LIN {X 0,Y 698.249,Z 977.53,A -85,B 0,C 180,E1 3562.598,E2 3562.598} C_VEL
LIN {X 0,Y 698.325,Z 977.53,A -85,B 0,C 180,E1 3567.816,E2 3567.816} C_VEL
LIN {X 0,Y 698.444,Z 977.53,A -85,B 0,C 180,E1 3572.91,E2 3572.91} C_VEL
LIN {X 0,Y 698.552,Z 977.53,A -85,B 0,C 180,E1 3577.03,E2 3577.03} C_VEL
LIN {X 0,Y 698.572,Z 977.53,A -85,B 0,C 180,E1 3582.649,E2 3582.649} C_VEL
LIN {X 0,Y 698.411,Z 977.53,A -85,B 0,C 180,E1 3587.531,E2 3587.531} C_VEL
LIN {X 0,Y 698.656,Z 977.53,A -85,B 0,C 180,E1 3592.533,E2 3592.533} C_VEL
LIN {X 0,Y 698.798,Z 977.53,A -85,B 0,C 180,E1 3596.63,E2 3596.63} C_VEL
LIN {X 0,Y 700.664,Z 990.787,A -85,B 0,C 180,E1 3596.832,E2 3596.832} C_VEL
LIN {X 0,Y 700.6,Z 1043.986,A -85,B 0,C 180,E1 3597.491,E2 3597.491} C_VEL
LIN {X 0,Y 700.227,Z 1071.881,A -85,B 0,C 180,E1 3598.304,E2 3598.304} C_VEL
LIN {X 0,Y 699.823,Z 1097.341,A -85,B 0,C 180,E1 3599.544,E2 3599.544} C_VEL
LIN {X 0,Y 699.493,Z 1119.031,A -85,B 0,C 180,E1 3601.095,E2 3601.095} C_VEL
LIN {X 0,Y 699.241,Z 1137.078,A -85,B 0,C 180,E1 3602.959,E2 3602.959} C_VEL
LIN {X 0,Y 699.113,Z 1150.198,A -85,B 0,C 180,E1 3604.982,E2 3604.982} C_VEL
LIN {X 0,Y 699.023,Z 1157.754,A -85,B 0,C 180,E1 3606.855,E2 3606.855} C_VEL
LIN {X 0,Y 698.935,Z 1161.69,A -85,B 0,C 180,E1 3608.737,E2 3608.737} C_VEL
LIN {X 0,Y 698.932,Z 1161.598,A -85,B 0,C 180,E1 3611.259,E2 3611.259} C_VEL
LIN {X 0,Y 699.047,Z 1156.293,A -85,B 0,C 180,E1 3613.499,E2 3613.499} C_VEL
LIN {X 0,Y 699.09,Z 1145.799,A -85,B 0,C 180,E1 3615.702,E2 3615.702} C_VEL
LIN {X 0,Y 699.304,Z 1129.473,A -85,B 0,C 180,E1 3617.829,E2 3617.829} C_VEL
LIN {X 0,Y 699.637,Z 1108.274,A -85,B 0,C 180,E1 3619.654,E2 3619.654} C_VEL
LIN {X 0,Y 700.068,Z 1082.113,A -85,B 0,C 180,E1 3621.168,E2 3621.168} C_VEL
LIN {X 0,Y 700.436,Z 1054.54,A -85,B 0,C 180,E1 3622.169,E2 3622.169} C_VEL
LIN {X 0,Y 700.63,Z 1024.887,A -85,B 0,C 180,E1 3622.707,E2 3622.707} C_VEL
LIN {X 0,Y 699.655,Z 981.842,A -85,B 0,C 180,E1 3623.185,E2 3623.185} C_VEL
LIN {X 0,Y 698.753,Z 977.53,A -85,B 0,C 180,E1 3623.298,E2 3623.298} C_VEL
LIN {X 0,Y 698.38,Z 977.53,A -85,B 0,C 180,E1 3628.518,E2 3628.518} C_VEL
LIN {X 0,Y 698.358,Z 977.53,A -85,B 0,C 180,E1 3632.856,E2 3632.856} C_VEL
LIN {X 0,Y 698.369,Z 977.53,A -85,B 0,C 180,E1 3637.416,E2 3637.416} C_VEL
LIN {X 0,Y 698.407,Z 977.53,A -85,B 0,C 180,E1 3642.459,E2 3642.459} C_VEL
LIN {X 0,Y 698.22,Z 977.53,A -85,B 0,C 180,E1 3647.712,E2 3647.712} C_VEL
LIN {X 0,Y 698.256,Z 977.53,A -85,B 0,C 180,E1 3652.575,E2 3652.575} C_VEL
LIN {X 0,Y 698.326,Z 977.53,A -85,B 0,C 180,E1 3657.811,E2 3657.811} C_VEL
LIN {X 0,Y 698.438,Z 977.53,A -85,B 0,C 180,E1 3662.89,E2 3662.89} C_VEL
LIN {X 0,Y 698.526,Z 977.53,A -85,B 0,C 180,E1 3667.011,E2 3667.011} C_VEL
LIN {X 0,Y 698.583,Z 977.53,A -85,B 0,C 180,E1 3672.635,E2 3672.635} C_VEL
LIN {X 0,Y 698.447,Z 977.53,A -85,B 0,C 180,E1 3677.502,E2 3677.502} C_VEL
LIN {X 0,Y 698.678,Z 977.53,A -85,B 0,C 180,E1 3682.517,E2 3682.517} C_VEL
LIN {X 0,Y 698.759,Z 977.53,A -85,B 0,C 180,E1 3687.509,E2 3687.509} C_VEL
LIN {X 0,Y 698.622,Z 977.53,A -85,B 0,C 180,E1 3692.48,E2 3692.48} C_VEL
LIN {X 0,Y 698.586,Z 977.53,A -85,B 0,C 180,E1 3696.22,E2 3696.22} C_VEL
LIN {X 0,Y 698.52,Z 977.53,A -85,B 0,C 180,E1 3701.252,E2 3701.252} C_VEL
LIN {X 0,Y 698.586,Z 977.53,A -85,B 0,C 180,E1 3706.372,E2 3706.372} C_VEL
LIN {X 0,Y 698.467,Z 977.53,A -85,B 0,C 180,E1 3711.635,E2 3711.635} C_VEL
LIN {X 0,Y 698.436,Z 977.53,A -85,B 0,C 180,E1 3715.709,E2 3715.709} C_VEL
LIN {X 0,Y 698.354,Z 977.53,A -85,B 0,C 180,E1 3719.93,E2 3719.93} C_VEL
LIN {X 0,Y 698.333,Z 977.53,A -85,B 0,C 180,E1 3724.453,E2 3724.453} C_VEL
LIN {X 0,Y 698.296,Z 977.53,A -85,B 0,C 180,E1 3728.99,E2 3728.99} C_VEL
LIN {X 0,Y 698.43,Z 977.53,A -85,B 0,C 180,E1 3734.274,E2 3734.274} C_VEL
LIN {X 0,Y 698.275,Z 977.53,A -85,B 0,C 180,E1 3739.411,E2 3739.411} C_VEL
LIN {X 0,Y 698.261,Z 977.53,A -85,B 0,C 180,E1 3744.126,E2 3744.126} C_VEL
LIN {X 0,Y 698.368,Z 977.53,A -85,B 0,C 180,E1 3748.612,E2 3748.612} C_VEL
LIN {X 0,Y 698.567,Z 977.53,A -85,B 0,C 180,E1 3754.283,E2 3754.283} C_VEL
LIN {X 0,Y 698.639,Z 977.53,A -85,B 0,C 180,E1 3754.865,E2 3754.865} C_VEL
LIN {X 0,Y 704.591,Z 996.788,A -85,B 0,C 180,E1 3755.324,E2 3755.324} C_VEL
LIN {X 0,Y 704.196,Z 1037.732,A -85,B 0,C 180,E1 3756.085,E2 3756.085} C_VEL
LIN {X 0,Y 703.296,Z 1074.948,A -85,B 0,C 180,E1 3757.243,E2 3757.243} C_VEL
LIN {X 0,Y 702.251,Z 1111.428,A -85,B 0,C 180,E1 3758.889,E2 3758.889} C_VEL
LIN {X 0,Y 701.238,Z 1144.866,A -85,B 0,C 180,E1 3760.94,E2 3760.94} C_VEL
LIN {X 0,Y 700.351,Z 1174.512,A -85,B 0,C 180,E1 3763.334,E2 3763.334} C_VEL
LIN {X 0,Y 699.676,Z 1200.165,A -85,B 0,C 180,E1 3766.051,E2 3766.051} C_VEL
LIN {X 0,Y 699.244,Z 1221.384,A -85,B 0,C 180,E1 3769.062,E2 3769.062} C_VEL
LIN {X 0,Y 699.071,Z 1237.084,A -85,B 0,C 180,E1 3772.206,E2 3772.206} C_VEL
LIN {X 0,Y 698.964,Z 1246.264,A -85,B 0,C 180,E1 3775.017,E2 3775.017} C_VEL
LIN {X 0,Y 698.927,Z 1250.943,A -85,B 0,C 180,E1 3777.506,E2 3777.506} C_VEL
LIN {X 0,Y 698.887,Z 1252.497,A -85,B 0,C 180,E1 3779.991,E2 3779.991} C_VEL
LIN {X 0,Y 698.948,Z 1250.844,A -85,B 0,C 180,E1 3782.476,E2 3782.476} C_VEL
LIN {X 0,Y 699.001,Z 1244.41,A -85,B 0,C 180,E1 3785.588,E2 3785.588} C_VEL
LIN {X 0,Y 699.048,Z 1232.688,A -85,B 0,C 180,E1 3788.717,E2 3788.717} C_VEL
LIN {X 0,Y 699.377,Z 1214.934,A -85,B 0,C 180,E1 3791.867,E2 3791.867} C_VEL
LIN {X 0,Y 699.823,Z 1192.335,A -85,B 0,C 180,E1 3794.772,E2 3794.772} C_VEL
LIN {X 0,Y 696.246,Z 1182.329,A -85,B 0,C 180,E1 3795.917,E2 3795.917} C_VEL
LIN {X 0,Y 692.744,Z 1171.657,A -85,B 0,C 180,E1 3797.032,E2 3797.032} C_VEL
LIN {X 0,Y 693.801,Z 1140.2,A -85,B 0,C 180,E1 3799.52,E2 3799.52} C_VEL
LIN {X 0,Y 694.966,Z 1105.397,A -85,B 0,C 180,E1 3801.576,E2 3801.576} C_VEL
LIN {X 0,Y 696.116,Z 1067.835,A -85,B 0,C 180,E1 3803.183,E2 3803.183} C_VEL
LIN {X 0,Y 697.047,Z 1028.121,A -85,B 0,C 180,E1 3804.317,E2 3804.317} C_VEL
LIN {X 0,Y 696.867,Z 995.477,A -85,B 0,C 180,E1 3804.895,E2 3804.895} C_VEL
LIN {X 0,Y 690.399,Z 977.53,A -85,B 0,C 180,E1 3805.41,E2 3805.41} C_VEL
LIN {X 0,Y 690.4,Z 977.53,A -85,B 0,C 180,E1 3810.303,E2 3810.303} C_VEL
LIN {X 0,Y 690.417,Z 977.53,A -85,B 0,C 180,E1 3815.714,E2 3815.714} C_VEL
LIN {X 0,Y 690.242,Z 977.53,A -85,B 0,C 180,E1 3819.804,E2 3819.804} C_VEL
LIN {X 0,Y 690.201,Z 977.53,A -85,B 0,C 180,E1 3824.611,E2 3824.611} C_VEL
LIN {X 0,Y 690.209,Z 977.53,A -85,B 0,C 180,E1 3828.814,E2 3828.814} C_VEL
LIN {X 0,Y 690.525,Z 977.53,A -85,B 0,C 180,E1 3834.259,E2 3834.259} C_VEL
LIN {X 0,Y 690.336,Z 977.53,A -85,B 0,C 180,E1 3839.686,E2 3839.686} C_VEL
LIN {X 0,Y 690.417,Z 977.584,A -85,B 0,C 180,E1 3842.029,E2 3842.029} C_VEL
LIN {X 0,Y 694.054,Z 987.272,A -85,B 0,C 180,E1 3842.718,E2 3842.718} C_VEL
LIN {X 0,Y 700.633,Z 994.826,A -85,B 0,C 180,E1 3843.899,E2 3843.899} C_VEL
LIN {X 0,Y 700.298,Z 999.146,A -85,B 0,C 180,E1 3844.205,E2 3844.205} C_VEL
LIN {X 0,Y 697.744,Z 1009.008,A -85,B 0,C 180,E1 3844.567,E2 3844.567} C_VEL
LIN {X 0,Y 697.181,Z 1078.924,A -85,B 0,C 180,E1 3845.446,E2 3845.446} C_VEL
LIN {X 0,Y 696.429,Z 1117.843,A -85,B 0,C 180,E1 3846.435,E2 3846.435} C_VEL
LIN {X 0,Y 695.282,Z 1155.762,A -85,B 0,C 180,E1 3847.911,E2 3847.911} C_VEL
LIN {X 0,Y 694.12,Z 1191.102,A -85,B 0,C 180,E1 3849.839,E2 3849.839} C_VEL
LIN {X 0,Y 692.969,Z 1223.117,A -85,B 0,C 180,E1 3852.18,E2 3852.18} C_VEL
LIN {X 0,Y 692.08,Z 1250.219,A -85,B 0,C 180,E1 3854.774,E2 3854.774} C_VEL
LIN {X 0,Y 691.534,Z 1273.012,A -85,B 0,C 180,E1 3857.67,E2 3857.67} C_VEL
LIN {X 0,Y 691.198,Z 1289.555,A -85,B 0,C 180,E1 3860.48,E2 3860.48} C_VEL
LIN {X 0,Y 691.049,Z 1302.604,A -85,B 0,C 180,E1 3863.712,E2 3863.712} C_VEL
LIN {X 0,Y 691.004,Z 1308.965,A -85,B 0,C 180,E1 3866.234,E2 3866.234} C_VEL
LIN {X 0,Y 691.014,Z 1312.108,A -85,B 0,C 180,E1 3868.749,E2 3868.749} C_VEL
LIN {X 0,Y 690.994,Z 1312.099,A -85,B 0,C 180,E1 3871.262,E2 3871.262} C_VEL
LIN {X 0,Y 691.006,Z 1307.534,A -85,B 0,C 180,E1 3874.464,E2 3874.464} C_VEL
LIN {X 0,Y 691.174,Z 1296.933,A -85,B 0,C 180,E1 3877.881,E2 3877.881} C_VEL
LIN {X 0,Y 691.431,Z 1281.1,A -85,B 0,C 180,E1 3881.061,E2 3881.061} C_VEL
LIN {X 0,Y 691.888,Z 1259.84,A -85,B 0,C 180,E1 3884.108,E2 3884.108} C_VEL
LIN {X 0,Y 692.673,Z 1234.009,A -85,B 0,C 180,E1 3886.855,E2 3886.855} C_VEL
LIN {X 0,Y 693.688,Z 1204.373,A -85,B 0,C 180,E1 3889.271,E2 3889.271} C_VEL
LIN {X 0,Y 694.806,Z 1170.678,A -85,B 0,C 180,E1 3891.348,E2 3891.348} C_VEL
LIN {X 0,Y 695.991,Z 1133.36,A -85,B 0,C 180,E1 3893.029,E2 3893.029} C_VEL
LIN {X 0,Y 696.975,Z 1094.227,A -85,B 0,C 180,E1 3894.224,E2 3894.224} C_VEL
LIN {X 0,Y 697.524,Z 1054.281,A -85,B 0,C 180,E1 3894.928,E2 3894.928} C_VEL
LIN {X 0,Y 697.79,Z 1008.208,A -85,B 0,C 180,E1 3895.492,E2 3895.492} C_VEL
LIN {X 0,Y 700.714,Z 996.51,A -85,B 0,C 180,E1 3895.944,E2 3895.944} C_VEL
LIN {X 0,Y 698.106,Z 991.717,A -85,B 0,C 180,E1 3896.672,E2 3896.672} C_VEL
LIN {X 0,Y 692.741,Z 985.09,A -85,B 0,C 180,E1 3897.48,E2 3897.48} C_VEL
LIN {X 0,Y 690.418,Z 977.53,A -85,B 0,C 180,E1 3898.047,E2 3898.047} C_VEL
LIN {X 0,Y 690.399,Z 977.53,A -85,B 0,C 180,E1 3903.284,E2 3903.284} C_VEL
LIN {X 0,Y 690.433,Z 977.53,A -85,B 0,C 180,E1 3907.923,E2 3907.923} C_VEL
LIN {X 0,Y 690.497,Z 977.53,A -85,B 0,C 180,E1 3913.62,E2 3913.62} C_VEL
LIN {X 0,Y 690.271,Z 977.53,A -85,B 0,C 180,E1 3918.828,E2 3918.828} C_VEL
LIN {X 0,Y 690.331,Z 977.53,A -85,B 0,C 180,E1 3924.316,E2 3924.316} C_VEL
LIN {X 0,Y 690.414,Z 977.53,A -85,B 0,C 180,E1 3929.697,E2 3929.697} C_VEL
LIN {X 0,Y 690.611,Z 977.53,A -85,B 0,C 180,E1 3934.116,E2 3934.116} C_VEL
LIN {X 0,Y 690.58,Z 977.53,A -85,B 0,C 180,E1 3939.459,E2 3939.459} C_VEL
LIN {X 0,Y 690.604,Z 977.53,A -85,B 0,C 180,E1 3944.746,E2 3944.746} C_VEL
LIN {X 0,Y 690.737,Z 977.53,A -85,B 0,C 180,E1 3949.903,E2 3949.903} C_VEL
LIN {X 0,Y 690.735,Z 977.53,A -85,B 0,C 180,E1 3954.976,E2 3954.976} C_VEL
LIN {X 0,Y 690.849,Z 977.53,A -85,B 0,C 180,E1 3956.418,E2 3956.418} C_VEL
LIN {X 0,Y 693.134,Z 991.243,A -85,B 0,C 180,E1 3956.645,E2 3956.645} C_VEL
LIN {X 0,Y 693.015,Z 1044.752,A -85,B 0,C 180,E1 3957.324,E2 3957.324} C_VEL
LIN {X 0,Y 692.601,Z 1073.222,A -85,B 0,C 180,E1 3958.168,E2 3958.168} C_VEL
LIN {X 0,Y 692.165,Z 1099.161,A -85,B 0,C 180,E1 3959.46,E2 3959.46} C_VEL
LIN {X 0,Y 691.726,Z 1121.136,A -85,B 0,C 180,E1 3961.107,E2 3961.107} C_VEL
LIN {X 0,Y 691.364,Z 1139.428,A -85,B 0,C 180,E1 3963.15,E2 3963.15} C_VEL
LIN {X 0,Y 691.177,Z 1152.174,A -85,B 0,C 180,E1 3965.355,E2 3965.355} C_VEL
LIN {X 0,Y 691.072,Z 1159.704,A -85,B 0,C 180,E1 3967.568,E2 3967.568} C_VEL
LIN {X 0,Y 691.034,Z 1162.385,A -85,B 0,C 180,E1 3970.111,E2 3970.111} C_VEL
LIN {X 0,Y 691.151,Z 1158.995,A -85,B 0,C 180,E1 3972.672,E2 3972.672} C_VEL
LIN {X 0,Y 691.243,Z 1150.473,A -85,B 0,C 180,E1 3974.933,E2 3974.933} C_VEL
LIN {X 0,Y 691.363,Z 1136.614,A -85,B 0,C 180,E1 3977.12,E2 3977.12} C_VEL
LIN {X 0,Y 691.742,Z 1118.326,A -85,B 0,C 180,E1 3979.023,E2 3979.023} C_VEL
LIN {X 0,Y 692.116,Z 1095.401,A -85,B 0,C 180,E1 3980.651,E2 3980.651} C_VEL
LIN {X 0,Y 692.679,Z 1069.013,A -85,B 0,C 180,E1 3981.881,E2 3981.881} C_VEL
LIN {X 0,Y 692.893,Z 1040.067,A -85,B 0,C 180,E1 3982.663,E2 3982.663} C_VEL
LIN {X 0,Y 692.216,Z 983.619,A -85,B 0,C 180,E1 3983.346,E2 3983.346} C_VEL
LIN {X 0,Y 690.826,Z 977.53,A -85,B 0,C 180,E1 3983.517,E2 3983.517} C_VEL
LIN {X 0,Y 690.461,Z 977.53,A -85,B 0,C 180,E1 3988.875,E2 3988.875} C_VEL
LIN {X 0,Y 690.394,Z 977.53,A -85,B 0,C 180,E1 3993.476,E2 3993.476} C_VEL
LIN {X 0,Y 690.447,Z 977.53,A -85,B 0,C 180,E1 3997.921,E2 3997.921} C_VEL
LIN {X 0,Y 690.507,Z 977.53,A -85,B 0,C 180,E1 4003.593,E2 4003.593} C_VEL
LIN {X 0,Y 690.272,Z 977.53,A -85,B 0,C 180,E1 4008.803,E2 4008.803} C_VEL
LIN {X 0,Y 690.323,Z 977.53,A -85,B 0,C 180,E1 4013.647,E2 4013.647} C_VEL
LIN {X 0,Y 690.434,Z 977.53,A -85,B 0,C 180,E1 4018.867,E2 4018.867} C_VEL
LIN {X 0,Y 690.586,Z 977.53,A -85,B 0,C 180,E1 4024.113,E2 4024.113} C_VEL
LIN {X 0,Y 690.567,Z 977.53,A -85,B 0,C 180,E1 4029.441,E2 4029.441} C_VEL
LIN {X 0,Y 690.654,Z 977.53,A -85,B 0,C 180,E1 4034.88,E2 4034.88} C_VEL
LIN {X 0,Y 690.758,Z 977.53,A -85,B 0,C 180,E1 4039.887,E2 4039.887} C_VEL
LIN {X 0,Y 690.725,Z 977.53,A -85,B 0,C 180,E1 4044.96,E2 4044.96} C_VEL
LIN {X 0,Y 690.796,Z 977.53,A -85,B 0,C 180,E1 4049.994,E2 4049.994} C_VEL
LIN {X 0,Y 690.911,Z 977.53,A -85,B 0,C 180,E1 4055.027,E2 4055.027} C_VEL
LIN {X 0,Y 690.64,Z 977.53,A -85,B 0,C 180,E1 4060.103,E2 4060.103} C_VEL
LIN {X 0,Y 690.634,Z 977.53,A -85,B 0,C 180,E1 4065.259,E2 4065.259} C_VEL
LIN {X 0,Y 690.61,Z 977.53,A -85,B 0,C 180,E1 4070.546,E2 4070.546} C_VEL
LIN {X 0,Y 690.511,Z 977.53,A -85,B 0,C 180,E1 4076.026,E2 4076.026} C_VEL
LIN {X 0,Y 690.44,Z 977.53,A -85,B 0,C 180,E1 4081.134,E2 4081.134} C_VEL
LIN {X 0,Y 690.451,Z 977.53,A -85,B 0,C 180,E1 4086.33,E2 4086.33} C_VEL
LIN {X 0,Y 690.418,Z 977.53,A -85,B 0,C 180,E1 4091.732,E2 4091.732} C_VEL
LIN {X 0,Y 690.369,Z 977.53,A -85,B 0,C 180,E1 4096.402,E2 4096.402} C_VEL
LIN {X 0,Y 690.345,Z 977.53,A -85,B 0,C 180,E1 4102.192,E2 4102.192} C_VEL
LIN {X 0,Y 690.347,Z 977.53,A -85,B 0,C 180,E1 4106.714,E2 4106.714} C_VEL
LIN {X 0,Y 690.468,Z 977.53,A -85,B 0,C 180,E1 4111.368,E2 4111.368} C_VEL
LIN {X 0,Y 690.701,Z 977.53,A -85,B 0,C 180,E1 4114.564,E2 4114.564} C_VEL
LIN {X 0,Y 697.426,Z 998.279,A -85,B 0,C 180,E1 4115.074,E2 4115.074} C_VEL
LIN {X 0,Y 696.954,Z 1038.128,A -85,B 0,C 180,E1 4115.832,E2 4115.832} C_VEL
LIN {X 0,Y 695.918,Z 1075.817,A -85,B 0,C 180,E1 4117.023,E2 4117.023} C_VEL
LIN {X 0,Y 694.785,Z 1111.418,A -85,B 0,C 180,E1 4118.651,E2 4118.651} C_VEL
LIN {X 0,Y 693.641,Z 1145.022,A -85,B 0,C 180,E1 4120.734,E2 4120.734} C_VEL
LIN {X 0,Y 692.632,Z 1174.504,A -85,B 0,C 180,E1 4123.143,E2 4123.143} C_VEL
LIN {X 0,Y 691.853,Z 1200.159,A -85,B 0,C 180,E1 4125.89,E2 4125.89} C_VEL
LIN {X 0,Y 691.393,Z 1221.379,A -85,B 0,C 180,E1 4128.936,E2 4128.936} C_VEL
LIN {X 0,Y 691.176,Z 1237.082,A -85,B 0,C 180,E1 4132.117,E2 4132.117} C_VEL
LIN {X 0,Y 691.059,Z 1246.263,A -85,B 0,C 180,E1 4134.96,E2 4134.96} C_VEL
LIN {X 0,Y 691.048,Z 1250.943,A -85,B 0,C 180,E1 4137.478,E2 4137.478} C_VEL
LIN {X 0,Y 690.989,Z 1252.497,A -85,B 0,C 180,E1 4139.991,E2 4139.991} C_VEL
LIN {X 0,Y 691.07,Z 1250.844,A -85,B 0,C 180,E1 4142.504,E2 4142.504} C_VEL
LIN {X 0,Y 691.11,Z 1244.411,A -85,B 0,C 180,E1 4145.652,E2 4145.652} C_VEL
LIN {X 0,Y 691.175,Z 1232.69,A -85,B 0,C 180,E1 4148.817,E2 4148.817} C_VEL
LIN {X 0,Y 691.536,Z 1214.935,A -85,B 0,C 180,E1 4152.004,E2 4152.004} C_VEL
LIN {X 0,Y 692.059,Z 1192.736,A -85,B 0,C 180,E1 4154.897,E2 4154.897} C_VEL
LIN {X 0,Y 692.744,Z 1171.657,A -85,B 0,C 180,E1 4157.032,E2 4157.032} C_VEL
LIN {X 0,Y 689.415,Z 1160.444,A -85,B 0,C 180,E1 4158.114,E2 4158.114} C_VEL
LIN {X 0,Y 685.964,Z 1148.483,A -85,B 0,C 180,E1 4159.145,E2 4159.145} C_VEL
LIN {X 0,Y 687.188,Z 1114.694,A -85,B 0,C 180,E1 4161.323,E2 4161.323} C_VEL
LIN {X 0,Y 688.488,Z 1078.679,A -85,B 0,C 180,E1 4163.032,E2 4163.032} C_VEL
LIN {X 0,Y 689.598,Z 1040.14,A -85,B 0,C 180,E1 4164.298,E2 4164.298} C_VEL
LIN {X 0,Y 690.337,Z 1001.799,A -85,B 0,C 180,E1 4165.059,E2 4165.059} C_VEL
LIN {X 0,Y 686.176,Z 988.352,A -85,B 0,C 180,E1 4165.395,E2 4165.395} C_VEL
LIN {X 0,Y 682.476,Z 977.53,A -85,B 0,C 180,E1 4165.706,E2 4165.706} C_VEL
LIN {X 0,Y 682.498,Z 977.53,A -85,B 0,C 180,E1 4170.692,E2 4170.692} C_VEL
LIN {X 0,Y 682.505,Z 977.53,A -85,B 0,C 180,E1 4175.241,E2 4175.241} C_VEL
LIN {X 0,Y 682.319,Z 977.53,A -85,B 0,C 180,E1 4180.075,E2 4180.075} C_VEL
LIN {X 0,Y 682.306,Z 977.53,A -85,B 0,C 180,E1 4185.268,E2 4185.268} C_VEL
LIN {X 0,Y 682.316,Z 977.53,A -85,B 0,C 180,E1 4189.915,E2 4189.915} C_VEL
LIN {X 0,Y 682.588,Z 977.53,A -85,B 0,C 180,E1 4195.195,E2 4195.195} C_VEL
LIN {X 0,Y 682.43,Z 977.53,A -85,B 0,C 180,E1 4200.766,E2 4200.766} C_VEL
LIN {X 0,Y 682.52,Z 977.629,A -85,B 0,C 180,E1 4201.762,E2 4201.762} C_VEL
LIN {X 0,Y 687.188,Z 991.103,A -85,B 0,C 180,E1 4202.586,E2 4202.586} C_VEL
LIN {X 0,Y 695.436,Z 1000.467,A -85,B 0,C 180,E1 4203.629,E2 4203.629} C_VEL
LIN {X 0,Y 690.509,Z 1020.031,A -85,B 0,C 180,E1 4204.41,E2 4204.41} C_VEL
LIN {X 0,Y 689.983,Z 1078.852,A -85,B 0,C 180,E1 4205.172,E2 4205.172} C_VEL
LIN {X 0,Y 689.124,Z 1119.013,A -85,B 0,C 180,E1 4206.209,E2 4206.209} C_VEL
LIN {X 0,Y 687.822,Z 1157.318,A -85,B 0,C 180,E1 4207.734,E2 4207.734} C_VEL
LIN {X 0,Y 686.529,Z 1192.516,A -85,B 0,C 180,E1 4209.699,E2 4209.699} C_VEL
LIN {X 0,Y 685.234,Z 1225.056,A -85,B 0,C 180,E1 4212.139,E2 4212.139} C_VEL
LIN {X 0,Y 684.285,Z 1251.688,A -85,B 0,C 180,E1 4214.761,E2 4214.761} C_VEL
LIN {X 0,Y 683.657,Z 1275.197,A -85,B 0,C 180,E1 4217.851,E2 4217.851} C_VEL
LIN {X 0,Y 683.255,Z 1292.852,A -85,B 0,C 180,E1 4221.075,E2 4221.075} C_VEL
LIN {X 0,Y 683.168,Z 1304.52,A -85,B 0,C 180,E1 4224.278,E2 4224.278} C_VEL
LIN {X 0,Y 683.094,Z 1310.934,A -85,B 0,C 180,E1 4227.463,E2 4227.463} C_VEL
LIN {X 0,Y 683.054,Z 1312.5,A -85,B 0,C 180,E1 4230.006,E2 4230.006} C_VEL
LIN {X 0,Y 683.105,Z 1310.918,A -85,B 0,C 180,E1 4232.549,E2 4232.549} C_VEL
LIN {X 0,Y 683.184,Z 1304.482,A -85,B 0,C 180,E1 4235.734,E2 4235.734} C_VEL
LIN {X 0,Y 683.257,Z 1292.802,A -85,B 0,C 180,E1 4238.937,E2 4238.937} C_VEL
LIN {X 0,Y 683.669,Z 1275.113,A -85,B 0,C 180,E1 4242.161,E2 4242.161} C_VEL
LIN {X 0,Y 684.317,Z 1251.583,A -85,B 0,C 180,E1 4245.251,E2 4245.251} C_VEL
LIN {X 0,Y 685.207,Z 1224.908,A -85,B 0,C 180,E1 4247.875,E2 4247.875} C_VEL
LIN {X 0,Y 686.538,Z 1192.383,A -85,B 0,C 180,E1 4250.309,E2 4250.309} C_VEL
LIN {X 0,Y 687.872,Z 1157.065,A -85,B 0,C 180,E1 4252.276,E2 4252.276} C_VEL
LIN {X 0,Y 689.162,Z 1118.794,A -85,B 0,C 180,E1 4253.797,E2 4253.797} C_VEL
LIN {X 0,Y 690.016,Z 1080.405,A -85,B 0,C 180,E1 4254.796,E2 4254.796} C_VEL
LIN {X 0,Y 690.788,Z 1018.224,A -85,B 0,C 180,E1 4255.679,E2 4255.679} C_VEL
LIN {X 0,Y 695.452,Z 1000.442,A -85,B 0,C 180,E1 4256.371,E2 4256.371} C_VEL
LIN {X 0,Y 687.125,Z 991.022,A -85,B 0,C 180,E1 4257.421,E2 4257.421} C_VEL
LIN {X 0,Y 682.537,Z 977.53,A -85,B 0,C 180,E1 4258.248,E2 4258.248} C_VEL
LIN {X 0,Y 682.492,Z 977.53,A -85,B 0,C 180,E1 4263.721,E2 4263.721} C_VEL
LIN {X 0,Y 682.407,Z 977.53,A -85,B 0,C 180,E1 4269.021,E2 4269.021} C_VEL
LIN {X 0,Y 682.589,Z 977.53,A -85,B 0,C 180,E1 4273.493,E2 4273.493} C_VEL
LIN {X 0,Y 682.372,Z 977.53,A -85,B 0,C 180,E1 4279.034,E2 4279.034} C_VEL
LIN {X 0,Y 682.394,Z 977.53,A -85,B 0,C 180,E1 4283.18,E2 4283.18} C_VEL
LIN {X 0,Y 682.456,Z 977.53,A -85,B 0,C 180,E1 4287.815,E2 4287.815} C_VEL
LIN {X 0,Y 682.642,Z 977.53,A -85,B 0,C 180,E1 4292.621,E2 4292.621} C_VEL
LIN {X 0,Y 682.681,Z 977.53,A -85,B 0,C 180,E1 4297.844,E2 4297.844} C_VEL
LIN {X 0,Y 682.716,Z 977.53,A -85,B 0,C 180,E1 4303.242,E2 4303.242} C_VEL
LIN {X 0,Y 682.719,Z 977.53,A -85,B 0,C 180,E1 4308.488,E2 4308.488} C_VEL
LIN {X 0,Y 682.931,Z 977.53,A -85,B 0,C 180,E1 4313.64,E2 4313.64} C_VEL
LIN {X 0,Y 682.973,Z 977.53,A -85,B 0,C 180,E1 4316.193,E2 4316.193} C_VEL
LIN {X 0,Y 685.607,Z 992.291,A -85,B 0,C 180,E1 4316.459,E2 4316.459} C_VEL
LIN {X 0,Y 685.385,Z 1047.325,A -85,B 0,C 180,E1 4317.193,E2 4317.193} C_VEL
LIN {X 0,Y 684.976,Z 1074.563,A -85,B 0,C 180,E1 4318.028,E2 4318.028} C_VEL
LIN {X 0,Y 684.502,Z 1099.665,A -85,B 0,C 180,E1 4319.296,E2 4319.296} C_VEL
LIN {X 0,Y 684.012,Z 1121.752,A -85,B 0,C 180,E1 4320.961,E2 4320.961} C_VEL
LIN {X 0,Y 683.615,Z 1140.046,A -85,B 0,C 180,E1 4323.008,E2 4323.008} C_VEL
LIN {X 0,Y 683.403,Z 1152.32,A -85,B 0,C 180,E1 4325.097,E2 4325.097} C_VEL
LIN {X 0,Y 683.285,Z 1159.304,A -85,B 0,C 180,E1 4327.014,E2 4327.014} C_VEL
LIN {X 0,Y 683.166,Z 1162.654,A -85,B 0,C 180,E1 4328.94,E2 4328.94} C_VEL
LIN {X 0,Y 683.2,Z 1162.057,A -85,B 0,C 180,E1 4331.522,E2 4331.522} C_VEL
LIN {X 0,Y 683.322,Z 1156.392,A -85,B 0,C 180,E1 4333.799,E2 4333.799} C_VEL
LIN {X 0,Y 683.499,Z 1145.242,A -85,B 0,C 180,E1 4336.096,E2 4336.096} C_VEL
LIN {X 0,Y 683.764,Z 1128.428,A -85,B 0,C 180,E1 4338.249,E2 4338.249} C_VEL
LIN {X 0,Y 684.231,Z 1106.993,A -85,B 0,C 180,E1 4340.086,E2 4340.086} C_VEL
LIN {X 0,Y 684.746,Z 1081.609,A -85,B 0,C 180,E1 4341.544,E2 4341.544} C_VEL
LIN {X 0,Y 685.204,Z 1053.597,A -85,B 0,C 180,E1 4342.537,E2 4342.537} C_VEL
LIN {X 0,Y 685.395,Z 1021.633,A -85,B 0,C 180,E1 4343.083,E2 4343.083} C_VEL
LIN {X 0,Y 684.488,Z 984.303,A -85,B 0,C 180,E1 4343.53,E2 4343.53} C_VEL
LIN {X 0,Y 682.898,Z 977.53,A -85,B 0,C 180,E1 4343.664,E2 4343.664} C_VEL
LIN {X 0,Y 682.506,Z 977.53,A -85,B 0,C 180,E1 4349.244,E2 4349.244} C_VEL
LIN {X 0,Y 682.479,Z 977.53,A -85,B 0,C 180,E1 4354.756,E2 4354.756} C_VEL
LIN {X 0,Y 682.411,Z 977.53,A -85,B 0,C 180,E1 4360.092,E2 4360.092} C_VEL
LIN {X 0,Y 682.569,Z 977.53,A -85,B 0,C 180,E1 4365.272,E2 4365.272} C_VEL
LIN {X 0,Y 682.399,Z 977.53,A -85,B 0,C 180,E1 4371.009,E2 4371.009} C_VEL
LIN {X 0,Y 682.434,Z 977.53,A -85,B 0,C 180,E1 4376.276,E2 4376.276} C_VEL
LIN {X 0,Y 682.504,Z 977.53,A -85,B 0,C 180,E1 4380.756,E2 4380.756} C_VEL
LIN {X 0,Y 682.648,Z 977.53,A -85,B 0,C 180,E1 4385.522,E2 4385.522} C_VEL
LIN {X 0,Y 682.667,Z 977.53,A -85,B 0,C 180,E1 4390.546,E2 4390.546} C_VEL
LIN {X 0,Y 682.661,Z 977.53,A -85,B 0,C 180,E1 4395.862,E2 4395.862} C_VEL
LIN {X 0,Y 682.782,Z 977.53,A -85,B 0,C 180,E1 4401.057,E2 4401.057} C_VEL
LIN {X 0,Y 682.945,Z 977.53,A -85,B 0,C 180,E1 4406.178,E2 4406.178} C_VEL
LIN {X 0,Y 683.048,Z 977.53,A -85,B 0,C 180,E1 4411.265,E2 4411.265} C_VEL
LIN {X 0,Y 682.783,Z 977.53,A -85,B 0,C 180,E1 4416.365,E2 4416.365} C_VEL
LIN {X 0,Y 682.734,Z 977.53,A -85,B 0,C 180,E1 4421.516,E2 4421.516} C_VEL
LIN {X 0,Y 682.762,Z 977.53,A -85,B 0,C 180,E1 4426.763,E2 4426.763} C_VEL
LIN {X 0,Y 682.609,Z 977.53,A -85,B 0,C 180,E1 4432.164,E2 4432.164} C_VEL
LIN {X 0,Y 682.598,Z 977.53,A -85,B 0,C 180,E1 4437.378,E2 4437.378} C_VEL
LIN {X 0,Y 682.486,Z 977.53,A -85,B 0,C 180,E1 4442.463,E2 4442.463} C_VEL
LIN {X 0,Y 682.498,Z 977.53,A -85,B 0,C 180,E1 4446.934,E2 4446.934} C_VEL
LIN {X 0,Y 682.59,Z 977.53,A -85,B 0,C 180,E1 4452.893,E2 4452.893} C_VEL
LIN {X 0,Y 682.426,Z 977.53,A -85,B 0,C 180,E1 4458.225,E2 4458.225} C_VEL
LIN {X 0,Y 682.402,Z 977.53,A -85,B 0,C 180,E1 4463.157,E2 4463.157} C_VEL
LIN {X 0,Y 682.461,Z 977.53,A -85,B 0,C 180,E1 4467.794,E2 4467.794} C_VEL
LIN {X 0,Y 682.65,Z 977.53,A -85,B 0,C 180,E1 4472.594,E2 4472.594} C_VEL
LIN {X 0,Y 682.805,Z 977.53,A -85,B 0,C 180,E1 4474.252,E2 4474.252} C_VEL
LIN {X 0,Y 690.253,Z 999.239,A -85,B 0,C 180,E1 4474.811,E2 4474.811} C_VEL
LIN {X 0,Y 689.68,Z 1039.37,A -85,B 0,C 180,E1 4475.595,E2 4475.595} C_VEL
LIN {X 0,Y 688.54,Z 1077.349,A -85,B 0,C 180,E1 4476.826,E2 4476.826} C_VEL
LIN {X 0,Y 687.274,Z 1112.922,A -85,B 0,C 180,E1 4478.491,E2 4478.491} C_VEL
LIN {X 0,Y 686.047,Z 1145.255,A -85,B 0,C 180,E1 4480.53,E2 4480.53} C_VEL
LIN {X 0,Y 684.897,Z 1174.496,A -85,B 0,C 180,E1 4482.946,E2 4482.946} C_VEL
LIN {X 0,Y 684.063,Z 1200.152,A -85,B 0,C 180,E1 4485.726,E2 4485.726} C_VEL
LIN {X 0,Y 683.536,Z 1221.374,A -85,B 0,C 180,E1 4488.808,E2 4488.808} C_VEL
LIN {X 0,Y 683.296,Z 1237.079,A -85,B 0,C 180,E1 4492.025,E2 4492.025} C_VEL
LIN {X 0,Y 683.1,Z 1247.794,A -85,B 0,C 180,E1 4495.539,E2 4495.539} C_VEL
LIN {X 0,Y 683.04,Z 1252.112,A -85,B 0,C 180,E1 4498.72,E2 4498.72} C_VEL
LIN {X 0,Y 683.198,Z 1252.054,A -85,B 0,C 180,E1 4501.262,E2 4501.262} C_VEL
LIN {X 0,Y 683.15,Z 1247.635,A -85,B 0,C 180,E1 4504.443,E2 4504.443} C_VEL
LIN {X 0,Y 683.228,Z 1238.074,A -85,B 0,C 180,E1 4507.637,E2 4507.637} C_VEL
LIN {X 0,Y 683.523,Z 1222.863,A -85,B 0,C 180,E1 4510.851,E2 4510.851} C_VEL
LIN {X 0,Y 684.049,Z 1200.895,A -85,B 0,C 180,E1 4514.092,E2 4514.092} C_VEL
LIN {X 0,Y 684.896,Z 1175.49,A -85,B 0,C 180,E1 4516.869,E2 4516.869} C_VEL
LIN {X 0,Y 685.964,Z 1148.483,A -85,B 0,C 180,E1 4519.145,E2 4519.145} C_VEL
LIN {X 0,Y 682.599,Z 1136.033,A -85,B 0,C 180,E1 4520.137,E2 4520.137} C_VEL
LIN {X 0,Y 679.405,Z 1122.967,A -85,B 0,C 180,E1 4521.087,E2 4521.087} C_VEL
LIN {X 0,Y 680.825,Z 1087.99,A -85,B 0,C 180,E1 4522.902,E2 4522.902} C_VEL
LIN {X 0,Y 682.15,Z 1050.202,A -85,B 0,C 180,E1 4524.29,E2 4524.29} C_VEL
LIN {X 0,Y 683.052,Z 1012.114,A -85,B 0,C 180,E1 4525.179,E2 4525.179} C_VEL
LIN {X 0,Y 682.381,Z 999.189,A -85,B 0,C 180,E1 4525.41,E2 4525.41} C_VEL
LIN {X 0,Y 674.559,Z 977.53,A -85,B 0,C 180,E1 4525.995,E2 4525.995} C_VEL
LIN {X 0,Y 674.557,Z 977.53,A -85,B 0,C 180,E1 4531.407,E2 4531.407} C_VEL
LIN {X 0,Y 674.532,Z 977.53,A -85,B 0,C 180,E1 4536.041,E2 4536.041} C_VEL
LIN {X 0,Y 674.422,Z 977.53,A -85,B 0,C 180,E1 4540.641,E2 4540.641} C_VEL
LIN {X 0,Y 674.371,Z 977.53,A -85,B 0,C 180,E1 4545.953,E2 4545.953} C_VEL
LIN {X 0,Y 674.489,Z 977.53,A -85,B 0,C 180,E1 4551.029,E2 4551.029} C_VEL
LIN {X 0,Y 674.615,Z 977.53,A -85,B 0,C 180,E1 4556.181,E2 4556.181} C_VEL
LIN {X 0,Y 674.646,Z 977.985,A -85,B 0,C 180,E1 4561.505,E2 4561.505} C_VEL
LIN {X 0,Y 679.919,Z 994.336,A -85,B 0,C 180,E1 4562.504,E2 4562.504} C_VEL
LIN {X 0,Y 688.687,Z 1004.683,A -85,B 0,C 180,E1 4563.365,E2 4563.365} C_VEL
LIN {X 0,Y 683.434,Z 1024.696,A -85,B 0,C 180,E1 4564.17,E2 4564.17} C_VEL
LIN {X 0,Y 682.798,Z 1081.048,A -85,B 0,C 180,E1 4564.936,E2 4564.936} C_VEL
LIN {X 0,Y 681.799,Z 1120.523,A -85,B 0,C 180,E1 4565.989,E2 4565.989} C_VEL
LIN {X 0,Y 680.395,Z 1158.964,A -85,B 0,C 180,E1 4567.559,E2 4567.559} C_VEL
LIN {X 0,Y 678.897,Z 1195.04,A -85,B 0,C 180,E1 4569.629,E2 4569.629} C_VEL
LIN {X 0,Y 677.506,Z 1227.283,A -85,B 0,C 180,E1 4572.123,E2 4572.123} C_VEL
LIN {X 0,Y 676.412,Z 1254.468,A -85,B 0,C 180,E1 4574.911,E2 4574.911} C_VEL
LIN {X 0,Y 675.833,Z 1276.355,A -85,B 0,C 180,E1 4577.883,E2 4577.883} C_VEL
LIN {X 0,Y 675.378,Z 1292.846,A -85,B 0,C 180,E1 4580.97,E2 4580.97} C_VEL
LIN {X 0,Y 675.296,Z 1304.518,A -85,B 0,C 180,E1 4584.211,E2 4584.211} C_VEL
LIN {X 0,Y 675.195,Z 1310.937,A -85,B 0,C 180,E1 4587.433,E2 4587.433} C_VEL
LIN {X 0,Y 675.179,Z 1312.5,A -85,B 0,C 180,E1 4590.006,E2 4590.006} C_VEL
LIN {X 0,Y 675.205,Z 1310.922,A -85,B 0,C 180,E1 4592.578,E2 4592.578} C_VEL
LIN {X 0,Y 675.311,Z 1304.48,A -85,B 0,C 180,E1 4595.801,E2 4595.801} C_VEL
LIN {X 0,Y 675.379,Z 1292.796,A -85,B 0,C 180,E1 4599.042,E2 4599.042} C_VEL
LIN {X 0,Y 675.839,Z 1275.218,A -85,B 0,C 180,E1 4602.288,E2 4602.288} C_VEL
LIN {X 0,Y 676.603,Z 1251.583,A -85,B 0,C 180,E1 4605.429,E2 4605.429} C_VEL
LIN {X 0,Y 677.647,Z 1223.622,A -85,B 0,C 180,E1 4608.192,E2 4608.192} C_VEL
LIN {X 0,Y 679.051,Z 1191.985,A -85,B 0,C 180,E1 4610.569,E2 4610.569} C_VEL
LIN {X 0,Y 680.47,Z 1157.059,A -85,B 0,C 180,E1 4612.532,E2 4612.532} C_VEL
LIN {X 0,Y 681.889,Z 1118.401,A -85,B 0,C 180,E1 4614.08,E2 4614.08} C_VEL
LIN {X 0,Y 682.904,Z 1078.176,A -85,B 0,C 180,E1 4615.116,E2 4615.116} C_VEL
LIN {X 0,Y 683.537,Z 1023.62,A -85,B 0,C 180,E1 4615.883,E2 4615.883} C_VEL
LIN {X 0,Y 688.113,Z 1004.001,A -85,B 0,C 180,E1 4616.704,E2 4616.704} C_VEL
LIN {X 0,Y 678.838,Z 992.286,A -85,B 0,C 180,E1 4617.587,E2 4617.587} C_VEL
LIN {X 0,Y 674.671,Z 977.53,A -85,B 0,C 180,E1 4618.415,E2 4618.415} C_VEL
LIN {X 0,Y 674.598,Z 977.53,A -85,B 0,C 180,E1 4624.17,E2 4624.17} C_VEL
LIN {X 0,Y 674.527,Z 977.53,A -85,B 0,C 180,E1 4628.984,E2 4628.984} C_VEL
LIN {X 0,Y 674.67,Z 977.53,A -85,B 0,C 180,E1 4634.134,E2 4634.134} C_VEL
LIN {X 0,Y 674.494,Z 977.53,A -85,B 0,C 180,E1 4639.811,E2 4639.811} C_VEL
LIN {X 0,Y 674.452,Z 977.53,A -85,B 0,C 180,E1 4644.275,E2 4644.275} C_VEL
LIN {X 0,Y 674.552,Z 977.53,A -85,B 0,C 180,E1 4648.907,E2 4648.907} C_VEL
LIN {X 0,Y 674.713,Z 977.53,A -85,B 0,C 180,E1 4653.951,E2 4653.951} C_VEL
LIN {X 0,Y 674.752,Z 977.53,A -85,B 0,C 180,E1 4658.955,E2 4658.955} C_VEL
LIN {X 0,Y 674.791,Z 977.53,A -85,B 0,C 180,E1 4664.379,E2 4664.379} C_VEL
LIN {X 0,Y 674.891,Z 977.53,A -85,B 0,C 180,E1 4669.663,E2 4669.663} C_VEL
LIN {X 0,Y 674.932,Z 977.53,A -85,B 0,C 180,E1 4674.858,E2 4674.858} C_VEL
LIN {X 0,Y 675.034,Z 977.659,A -85,B 0,C 180,E1 4675.987,E2 4675.987} C_VEL
LIN {X 0,Y 678.035,Z 990.971,A -85,B 0,C 180,E1 4676.242,E2 4676.242} C_VEL
LIN {X 0,Y 677.814,Z 1048.659,A -85,B 0,C 180,E1 4677.032,E2 4677.032} C_VEL
LIN {X 0,Y 677.374,Z 1076.888,A -85,B 0,C 180,E1 4677.926,E2 4677.926} C_VEL
LIN {X 0,Y 676.819,Z 1102.769,A -85,B 0,C 180,E1 4679.288,E2 4679.288} C_VEL
LIN {X 0,Y 676.281,Z 1124.072,A -85,B 0,C 180,E1 4680.972,E2 4680.972} C_VEL
LIN {X 0,Y 675.84,Z 1141.88,A -85,B 0,C 180,E1 4683.043,E2 4683.043} C_VEL
LIN {X 0,Y 675.601,Z 1155.169,A -85,B 0,C 180,E1 4685.478,E2 4685.478} C_VEL
LIN {X 0,Y 675.379,Z 1161.965,A -85,B 0,C 180,E1 4687.745,E2 4687.745} C_VEL
LIN {X 0,Y 675.351,Z 1164.038,A -85,B 0,C 180,E1 4690.348,E2 4690.348} C_VEL
LIN {X 0,Y 675.475,Z 1160.007,A -85,B 0,C 180,E1 4692.971,E2 4692.971} C_VEL
LIN {X 0,Y 675.595,Z 1150.909,A -85,B 0,C 180,E1 4695.306,E2 4695.306} C_VEL
LIN {X 0,Y 675.894,Z 1136.41,A -85,B 0,C 180,E1 4697.528,E2 4697.528} C_VEL
LIN {X 0,Y 676.356,Z 1117.319,A -85,B 0,C 180,E1 4699.473,E2 4699.473} C_VEL
LIN {X 0,Y 676.834,Z 1093.923,A -85,B 0,C 180,E1 4701.098,E2 4701.098} C_VEL
LIN {X 0,Y 677.448,Z 1067.212,A -85,B 0,C 180,E1 4702.299,E2 4702.299} C_VEL
LIN {X 0,Y 677.675,Z 1038.517,A -85,B 0,C 180,E1 4703.035,E2 4703.035} C_VEL
LIN {X 0,Y 677.304,Z 987.072,A -85,B 0,C 180,E1 4703.682,E2 4703.682} C_VEL
LIN {X 0,Y 674.959,Z 977.53,A -85,B 0,C 180,E1 4703.897,E2 4703.897} C_VEL
LIN {X 0,Y 674.58,Z 977.53,A -85,B 0,C 180,E1 4709.622,E2 4709.622} C_VEL
LIN {X 0,Y 674.565,Z 977.53,A -85,B 0,C 180,E1 4714.171,E2 4714.171} C_VEL
LIN {X 0,Y 674.56,Z 977.53,A -85,B 0,C 180,E1 4718.98,E2 4718.98} C_VEL
LIN {X 0,Y 674.678,Z 977.53,A -85,B 0,C 180,E1 4724.132,E2 4724.132} C_VEL
LIN {X 0,Y 674.484,Z 977.53,A -85,B 0,C 180,E1 4729.809,E2 4729.809} C_VEL
LIN {X 0,Y 674.451,Z 977.53,A -85,B 0,C 180,E1 4734.251,E2 4734.251} C_VEL
LIN {X 0,Y 674.56,Z 977.53,A -85,B 0,C 180,E1 4738.885,E2 4738.885} C_VEL
LIN {X 0,Y 674.707,Z 977.53,A -85,B 0,C 180,E1 4743.946,E2 4743.946} C_VEL
LIN {X 0,Y 674.747,Z 977.53,A -85,B 0,C 180,E1 4748.936,E2 4748.936} C_VEL
LIN {X 0,Y 674.821,Z 977.53,A -85,B 0,C 180,E1 4754.362,E2 4754.362} C_VEL
LIN {X 0,Y 674.917,Z 977.53,A -85,B 0,C 180,E1 4759.647,E2 4759.647} C_VEL
LIN {X 0,Y 674.921,Z 977.53,A -85,B 0,C 180,E1 4764.842,E2 4764.842} C_VEL
LIN {X 0,Y 675.011,Z 977.53,A -85,B 0,C 180,E1 4769.994,E2 4769.994} C_VEL
LIN {X 0,Y 675.1,Z 977.53,A -85,B 0,C 180,E1 4775.145,E2 4775.145} C_VEL
LIN {X 0,Y 674.814,Z 977.53,A -85,B 0,C 180,E1 4780.342,E2 4780.342} C_VEL
LIN {X 0,Y 674.819,Z 977.53,A -85,B 0,C 180,E1 4785.625,E2 4785.625} C_VEL
LIN {X 0,Y 674.751,Z 977.53,A -85,B 0,C 180,E1 4791.051,E2 4791.051} C_VEL
LIN {X 0,Y 674.667,Z 977.53,A -85,B 0,C 180,E1 4796.685,E2 4796.685} C_VEL
LIN {X 0,Y 674.564,Z 977.53,A -85,B 0,C 180,E1 4801.389,E2 4801.389} C_VEL
LIN {X 0,Y 674.54,Z 977.53,A -85,B 0,C 180,E1 4806.025,E2 4806.025} C_VEL
LIN {X 0,Y 674.537,Z 977.53,A -85,B 0,C 180,E1 4810.643,E2 4810.643} C_VEL
LIN {X 0,Y 674.566,Z 977.53,A -85,B 0,C 180,E1 4815.948,E2 4815.948} C_VEL
LIN {X 0,Y 674.522,Z 977.53,A -85,B 0,C 180,E1 4821.017,E2 4821.017} C_VEL
LIN {X 0,Y 674.532,Z 977.53,A -85,B 0,C 180,E1 4826.208,E2 4826.208} C_VEL
LIN {X 0,Y 674.647,Z 977.53,A -85,B 0,C 180,E1 4831.851,E2 4831.851} C_VEL
LIN {X 0,Y 674.816,Z 977.53,A -85,B 0,C 180,E1 4833.94,E2 4833.94} C_VEL
LIN {X 0,Y 683.114,Z 1001.544,A -85,B 0,C 180,E1 4834.564,E2 4834.564} C_VEL
LIN {X 0,Y 682.43,Z 1041.107,A -85,B 0,C 180,E1 4835.367,E2 4835.367} C_VEL
LIN {X 0,Y 681.19,Z 1078.446,A -85,B 0,C 180,E1 4836.607,E2 4836.607} C_VEL
LIN {X 0,Y 679.779,Z 1114.426,A -85,B 0,C 180,E1 4838.327,E2 4838.327} C_VEL
LIN {X 0,Y 678.352,Z 1147.948,A -85,B 0,C 180,E1 4840.501,E2 4840.501} C_VEL
LIN {X 0,Y 677.139,Z 1177.972,A -85,B 0,C 180,E1 4843.08,E2 4843.08} C_VEL
LIN {X 0,Y 676.198,Z 1203.99,A -85,B 0,C 180,E1 4846.053,E2 4846.053} C_VEL
LIN {X 0,Y 675.637,Z 1223.248,A -85,B 0,C 180,E1 4849.002,E2 4849.002} C_VEL
LIN {X 0,Y 675.372,Z 1238.327,A -85,B 0,C 180,E1 4852.255,E2 4852.255} C_VEL
LIN {X 0,Y 675.204,Z 1247.793,A -85,B 0,C 180,E1 4855.486,E2 4855.486} C_VEL
LIN {X 0,Y 675.153,Z 1252.112,A -85,B 0,C 180,E1 4858.705,E2 4858.705} C_VEL
LIN {X 0,Y 675.326,Z 1252.055,A -85,B 0,C 180,E1 4861.276,E2 4861.276} C_VEL
LIN {X 0,Y 675.253,Z 1247.636,A -85,B 0,C 180,E1 4864.495,E2 4864.495} C_VEL
LIN {X 0,Y 675.343,Z 1238.077,A -85,B 0,C 180,E1 4867.727,E2 4867.727} C_VEL
LIN {X 0,Y 675.684,Z 1222.866,A -85,B 0,C 180,E1 4870.978,E2 4870.978} C_VEL
LIN {X 0,Y 676.26,Z 1200.897,A -85,B 0,C 180,E1 4874.258,E2 4874.258} C_VEL
LIN {X 0,Y 677.211,Z 1175.578,A -85,B 0,C 180,E1 4877.058,E2 4877.058} C_VEL
LIN {X 0,Y 678.421,Z 1145.857,A -85,B 0,C 180,E1 4879.562,E2 4879.562} C_VEL
LIN {X 0,Y 679.405,Z 1122.967,A -85,B 0,C 180,E1 4881.087,E2 4881.087} C_VEL
LIN {X 0,Y 676.337,Z 1109.448,A -85,B 0,C 180,E1 4881.997,E2 4881.997} C_VEL
LIN {X 0,Y 673.252,Z 1095.303,A -85,B 0,C 180,E1 4882.832,E2 4882.832} C_VEL
LIN {X 0,Y 674.699,Z 1056.986,A -85,B 0,C 180,E1 4884.356,E2 4884.356} C_VEL
LIN {X 0,Y 675.701,Z 1018.673,A -85,B 0,C 180,E1 4885.344,E2 4885.344} C_VEL
LIN {X 0,Y 675.169,Z 1001.313,A -85,B 0,C 180,E1 4885.652,E2 4885.652} C_VEL
LIN {X 0,Y 666.638,Z 977.53,A -85,B 0,C 180,E1 4886.265,E2 4886.265} C_VEL
LIN {X 0,Y 666.663,Z 977.53,A -85,B 0,C 180,E1 4891.503,E2 4891.503} C_VEL
LIN {X 0,Y 666.617,Z 977.53,A -85,B 0,C 180,E1 4896.211,E2 4896.211} C_VEL
LIN {X 0,Y 666.467,Z 977.53,A -85,B 0,C 180,E1 4901.395,E2 4901.395} C_VEL
LIN {X 0,Y 666.432,Z 977.53,A -85,B 0,C 180,E1 4907,E2 4907} C_VEL
LIN {X 0,Y 666.674,Z 977.53,A -85,B 0,C 180,E1 4912.679,E2 4912.679} C_VEL
LIN {X 0,Y 666.666,Z 977.53,A -85,B 0,C 180,E1 4917.215,E2 4917.215} C_VEL
LIN {X 0,Y 666.664,Z 977.54,A -85,B 0,C 180,E1 4921.199,E2 4921.199} C_VEL
LIN {X 0,Y 672.074,Z 996.263,A -85,B 0,C 180,E1 4922.336,E2 4922.336} C_VEL
LIN {X 0,Y 680.637,Z 1008.384,A -85,B 0,C 180,E1 4923.223,E2 4923.223} C_VEL
LIN {X 0,Y 676.166,Z 1025.286,A -85,B 0,C 180,E1 4923.916,E2 4923.916} C_VEL
LIN {X 0,Y 675.617,Z 1080.872,A -85,B 0,C 180,E1 4924.651,E2 4924.651} C_VEL
LIN {X 0,Y 674.538,Z 1120.683,A -85,B 0,C 180,E1 4925.72,E2 4925.72} C_VEL
LIN {X 0,Y 673.009,Z 1159.067,A -85,B 0,C 180,E1 4927.305,E2 4927.305} C_VEL
LIN {X 0,Y 671.412,Z 1194.096,A -85,B 0,C 180,E1 4929.328,E2 4929.328} C_VEL
LIN {X 0,Y 669.875,Z 1226.915,A -85,B 0,C 180,E1 4931.879,E2 4931.879} C_VEL
LIN {X 0,Y 668.664,Z 1254.461,A -85,B 0,C 180,E1 4934.732,E2 4934.732} C_VEL
LIN {X 0,Y 667.972,Z 1276.085,A -85,B 0,C 180,E1 4937.697,E2 4937.697} C_VEL
LIN {X 0,Y 667.511,Z 1292.84,A -85,B 0,C 180,E1 4940.863,E2 4940.863} C_VEL
LIN {X 0,Y 667.397,Z 1304.516,A -85,B 0,C 180,E1 4944.142,E2 4944.142} C_VEL
LIN {X 0,Y 667.315,Z 1310.939,A -85,B 0,C 180,E1 4947.403,E2 4947.403} C_VEL
LIN {X 0,Y 667.28,Z 1312.5,A -85,B 0,C 180,E1 4950.006,E2 4950.006} C_VEL
LIN {X 0,Y 667.292,Z 1310.754,A -85,B 0,C 180,E1 4952.741,E2 4952.741} C_VEL
LIN {X 0,Y 667.412,Z 1304.478,A -85,B 0,C 180,E1 4955.87,E2 4955.87} C_VEL
LIN {X 0,Y 667.512,Z 1292.79,A -85,B 0,C 180,E1 4959.149,E2 4959.149} C_VEL
LIN {X 0,Y 667.985,Z 1276.009,A -85,B 0,C 180,E1 4962.314,E2 4962.314} C_VEL
LIN {X 0,Y 668.786,Z 1252.97,A -85,B 0,C 180,E1 4965.445,E2 4965.445} C_VEL
LIN {X 0,Y 669.83,Z 1227.058,A -85,B 0,C 180,E1 4968.109,E2 4968.109} C_VEL
LIN {X 0,Y 671.442,Z 1194.056,A -85,B 0,C 180,E1 4970.673,E2 4970.673} C_VEL
LIN {X 0,Y 673.027,Z 1159.278,A -85,B 0,C 180,E1 4972.684,E2 4972.684} C_VEL
LIN {X 0,Y 674.562,Z 1121.723,A -85,B 0,C 180,E1 4974.244,E2 4974.244} C_VEL
LIN {X 0,Y 675.64,Z 1082.464,A -85,B 0,C 180,E1 4975.317,E2 4975.317} C_VEL
LIN {X 0,Y 676.012,Z 1035.582,A -85,B 0,C 180,E1 4975.969,E2 4975.969} C_VEL
LIN {X 0,Y 676.45,Z 1023.086,A -85,B 0,C 180,E1 4976.175,E2 4976.175} C_VEL
LIN {X 0,Y 680.212,Z 1006.947,A -85,B 0,C 180,E1 4976.852,E2 4976.852} C_VEL
LIN {X 0,Y 671.389,Z 994.904,A -85,B 0,C 180,E1 4977.657,E2 4977.657} C_VEL
LIN {X 0,Y 666.715,Z 977.53,A -85,B 0,C 180,E1 4978.682,E2 4978.682} C_VEL
LIN {X 0,Y 666.68,Z 977.53,A -85,B 0,C 180,E1 4983.065,E2 4983.065} C_VEL
LIN {X 0,Y 666.639,Z 977.53,A -85,B 0,C 180,E1 4987.866,E2 4987.866} C_VEL
LIN {X 0,Y 666.681,Z 977.53,A -85,B 0,C 180,E1 4993.359,E2 4993.359} C_VEL
LIN {X 0,Y 666.531,Z 977.53,A -85,B 0,C 180,E1 4998.774,E2 4998.774} C_VEL
LIN {X 0,Y 666.54,Z 977.53,A -85,B 0,C 180,E1 5003.784,E2 5003.784} C_VEL
LIN {X 0,Y 666.654,Z 977.53,A -85,B 0,C 180,E1 5008.496,E2 5008.496} C_VEL
LIN {X 0,Y 666.767,Z 977.53,A -85,B 0,C 180,E1 5012.98,E2 5012.98} C_VEL
LIN {X 0,Y 666.832,Z 977.53,A -85,B 0,C 180,E1 5017.289,E2 5017.289} C_VEL
LIN {X 0,Y 666.88,Z 977.53,A -85,B 0,C 180,E1 5022.831,E2 5022.831} C_VEL
LIN {X 0,Y 666.861,Z 977.53,A -85,B 0,C 180,E1 5028.211,E2 5028.211} C_VEL
LIN {X 0,Y 667.101,Z 977.53,A -85,B 0,C 180,E1 5033.489,E2 5033.489} C_VEL
LIN {X 0,Y 667.11,Z 977.53,A -85,B 0,C 180,E1 5035.743,E2 5035.743} C_VEL
LIN {X 0,Y 670.572,Z 993.13,A -85,B 0,C 180,E1 5036.056,E2 5036.056} C_VEL
LIN {X 0,Y 670.235,Z 1049.316,A -85,B 0,C 180,E1 5036.851,E2 5036.851} C_VEL
LIN {X 0,Y 669.764,Z 1078.225,A -85,B 0,C 180,E1 5037.781,E2 5037.781} C_VEL
LIN {X 0,Y 669.168,Z 1103.281,A -85,B 0,C 180,E1 5039.117,E2 5039.117} C_VEL
LIN {X 0,Y 668.568,Z 1124.7,A -85,B 0,C 180,E1 5040.821,E2 5040.821} C_VEL
LIN {X 0,Y 668.074,Z 1143.151,A -85,B 0,C 180,E1 5042.995,E2 5042.995} C_VEL
LIN {X 0,Y 667.786,Z 1155.321,A -85,B 0,C 180,E1 5045.216,E2 5045.216} C_VEL
LIN {X 0,Y 667.539,Z 1163.189,A -85,B 0,C 180,E1 5047.836,E2 5047.836} C_VEL
LIN {X 0,Y 667.517,Z 1164.929,A -85,B 0,C 180,E1 5050.471,E2 5050.471} C_VEL
LIN {X 0,Y 667.606,Z 1162.032,A -85,B 0,C 180,E1 5052.559,E2 5052.559} C_VEL
LIN {X 0,Y 667.803,Z 1152.931,A -85,B 0,C 180,E1 5055.148,E2 5055.148} C_VEL
LIN {X 0,Y 668.056,Z 1138.757,A -85,B 0,C 180,E1 5057.435,E2 5057.435} C_VEL
LIN {X 0,Y 668.535,Z 1120.731,A -85,B 0,C 180,E1 5059.366,E2 5059.366} C_VEL
LIN {X 0,Y 669.059,Z 1097.34,A -85,B 0,C 180,E1 5061.079,E2 5061.079} C_VEL
LIN {X 0,Y 669.785,Z 1070.999,A -85,B 0,C 180,E1 5062.342,E2 5062.342} C_VEL
LIN {X 0,Y 670.049,Z 1042.035,A -85,B 0,C 180,E1 5063.152,E2 5063.152} C_VEL
LIN {X 0,Y 669.602,Z 987.812,A -85,B 0,C 180,E1 5063.871,E2 5063.871} C_VEL
LIN {X 0,Y 667.031,Z 977.53,A -85,B 0,C 180,E1 5064.092,E2 5064.092} C_VEL
LIN {X 0,Y 666.628,Z 977.53,A -85,B 0,C 180,E1 5070.011,E2 5070.011} C_VEL
LIN {X 0,Y 666.597,Z 977.53,A -85,B 0,C 180,E1 5075.072,E2 5075.072} C_VEL
LIN {X 0,Y 666.608,Z 977.53,A -85,B 0,C 180,E1 5079.535,E2 5079.535} C_VEL
LIN {X 0,Y 666.672,Z 977.53,A -85,B 0,C 180,E1 5084.803,E2 5084.803} C_VEL
LIN {X 0,Y 666.591,Z 977.53,A -85,B 0,C 180,E1 5090.619,E2 5090.619} C_VEL
LIN {X 0,Y 666.55,Z 977.53,A -85,B 0,C 180,E1 5095.359,E2 5095.359} C_VEL
LIN {X 0,Y 666.639,Z 977.53,A -85,B 0,C 180,E1 5099.989,E2 5099.989} C_VEL
LIN {X 0,Y 666.768,Z 977.53,A -85,B 0,C 180,E1 5105.378,E2 5105.378} C_VEL
LIN {X 0,Y 666.81,Z 977.53,A -85,B 0,C 180,E1 5110.064,E2 5110.064} C_VEL
LIN {X 0,Y 666.898,Z 977.53,A -85,B 0,C 180,E1 5114.172,E2 5114.172} C_VEL
LIN {X 0,Y 666.995,Z 977.53,A -85,B 0,C 180,E1 5119.523,E2 5119.523} C_VEL
LIN {X 0,Y 667.032,Z 977.53,A -85,B 0,C 180,E1 5124.781,E2 5124.781} C_VEL
LIN {X 0,Y 667.111,Z 977.53,A -85,B 0,C 180,E1 5129.994,E2 5129.994} C_VEL
LIN {X 0,Y 667.208,Z 977.53,A -85,B 0,C 180,E1 5135.206,E2 5135.206} C_VEL
LIN {X 0,Y 666.901,Z 977.53,A -85,B 0,C 180,E1 5140.467,E2 5140.467} C_VEL
LIN {X 0,Y 666.901,Z 977.53,A -85,B 0,C 180,E1 5145.816,E2 5145.816} C_VEL
LIN {X 0,Y 666.809,Z 977.53,A -85,B 0,C 180,E1 5151.314,E2 5151.314} C_VEL
LIN {X 0,Y 666.744,Z 977.53,A -85,B 0,C 180,E1 5155.575,E2 5155.575} C_VEL
LIN {X 0,Y 666.64,Z 977.53,A -85,B 0,C 180,E1 5160.255,E2 5160.255} C_VEL
LIN {X 0,Y 666.611,Z 977.53,A -85,B 0,C 180,E1 5165.077,E2 5165.077} C_VEL
LIN {X 0,Y 666.611,Z 977.53,A -85,B 0,C 180,E1 5169.521,E2 5169.521} C_VEL
LIN {X 0,Y 666.65,Z 977.53,A -85,B 0,C 180,E1 5174.79,E2 5174.79} C_VEL
LIN {X 0,Y 666.589,Z 977.53,A -85,B 0,C 180,E1 5180.603,E2 5180.603} C_VEL
LIN {X 0,Y 666.545,Z 977.53,A -85,B 0,C 180,E1 5185.36,E2 5185.36} C_VEL
LIN {X 0,Y 666.635,Z 977.53,A -85,B 0,C 180,E1 5189.989,E2 5189.989} C_VEL
LIN {X 0,Y 666.915,Z 978.095,A -85,B 0,C 180,E1 5193.653,E2 5193.653} C_VEL
LIN {X 0,Y 675.885,Z 1004.223,A -85,B 0,C 180,E1 5194.32,E2 5194.32} C_VEL
LIN {X 0,Y 675.121,Z 1044.503,A -85,B 0,C 180,E1 5195.178,E2 5195.178} C_VEL
LIN {X 0,Y 673.707,Z 1083.681,A -85,B 0,C 180,E1 5196.552,E2 5196.552} C_VEL
LIN {X 0,Y 672.099,Z 1120.312,A -85,B 0,C 180,E1 5198.415,E2 5198.415} C_VEL
LIN {X 0,Y 670.527,Z 1153.37,A -85,B 0,C 180,E1 5200.694,E2 5200.694} C_VEL
LIN {X 0,Y 669.288,Z 1181.212,A -85,B 0,C 180,E1 5203.215,E2 5203.215} C_VEL
LIN {X 0,Y 668.363,Z 1205.196,A -85,B 0,C 180,E1 5206.054,E2 5206.054} C_VEL
LIN {X 0,Y 667.711,Z 1224.988,A -85,B 0,C 180,E1 5209.201,E2 5209.201} C_VEL
LIN {X 0,Y 667.487,Z 1239.471,A -85,B 0,C 180,E1 5212.491,E2 5212.491} C_VEL
LIN {X 0,Y 667.316,Z 1247.792,A -85,B 0,C 180,E1 5215.433,E2 5215.433} C_VEL
LIN {X 0,Y 667.253,Z 1252.112,A -85,B 0,C 180,E1 5218.69,E2 5218.69} C_VEL
LIN {X 0,Y 667.424,Z 1252.056,A -85,B 0,C 180,E1 5221.291,E2 5221.291} C_VEL
LIN {X 0,Y 667.356,Z 1247.637,A -85,B 0,C 180,E1 5224.548,E2 5224.548} C_VEL
LIN {X 0,Y 667.481,Z 1238.079,A -85,B 0,C 180,E1 5227.818,E2 5227.818} C_VEL
LIN {X 0,Y 667.836,Z 1222.87,A -85,B 0,C 180,E1 5231.109,E2 5231.109} C_VEL
LIN {X 0,Y 668.43,Z 1202.216,A -85,B 0,C 180,E1 5234.261,E2 5234.261} C_VEL
LIN {X 0,Y 669.508,Z 1175.79,A -85,B 0,C 180,E1 5237.24,E2 5237.24} C_VEL
LIN {X 0,Y 670.889,Z 1145.863,A -85,B 0,C 180,E1 5239.791,E2 5239.791} C_VEL
LIN {X 0,Y 672.337,Z 1113.198,A -85,B 0,C 180,E1 5241.905,E2 5241.905} C_VEL
LIN {X 0,Y 673.252,Z 1095.303,A -85,B 0,C 180,E1 5242.832,E2 5242.832} C_VEL
LIN {X 0,Y 669.88,Z 1085.966,A -85,B 0,C 180,E1 5243.394,E2 5243.394} C_VEL
LIN {X 0,Y 666.564,Z 1076.457,A -85,B 0,C 180,E1 5243.92,E2 5243.92} C_VEL
LIN {X 0,Y 667.934,Z 1037.18,A -85,B 0,C 180,E1 5245.181,E2 5245.181} C_VEL
LIN {X 0,Y 667.88,Z 1003.499,A -85,B 0,C 180,E1 5245.865,E2 5245.865} C_VEL
LIN {X 0,Y 658.742,Z 977.53,A -85,B 0,C 180,E1 5246.561,E2 5246.561} C_VEL
LIN {X 0,Y 658.761,Z 977.53,A -85,B 0,C 180,E1 5251.925,E2 5251.925} C_VEL
LIN {X 0,Y 658.699,Z 977.53,A -85,B 0,C 180,E1 5256.717,E2 5256.717} C_VEL
LIN {X 0,Y 658.524,Z 977.53,A -85,B 0,C 180,E1 5261.839,E2 5261.839} C_VEL
LIN {X 0,Y 658.491,Z 977.53,A -85,B 0,C 180,E1 5267.401,E2 5267.401} C_VEL
LIN {X 0,Y 658.772,Z 977.53,A -85,B 0,C 180,E1 5273.278,E2 5273.278} C_VEL
LIN {X 0,Y 658.72,Z 977.53,A -85,B 0,C 180,E1 5278.304,E2 5278.304} C_VEL
LIN {X 0,Y 658.75,Z 977.625,A -85,B 0,C 180,E1 5280.922,E2 5280.922} C_VEL
LIN {X 0,Y 664.703,Z 999.06,A -85,B 0,C 180,E1 5282.233,E2 5282.233} C_VEL
LIN {X 0,Y 672.407,Z 1011.419,A -85,B 0,C 180,E1 5283.109,E2 5283.109} C_VEL
LIN {X 0,Y 668.892,Z 1024.492,A -85,B 0,C 180,E1 5283.656,E2 5283.656} C_VEL
LIN {X 0,Y 668.231,Z 1079.813,A -85,B 0,C 180,E1 5284.396,E2 5284.396} C_VEL
LIN {X 0,Y 667.134,Z 1121.583,A -85,B 0,C 180,E1 5285.498,E2 5285.498} C_VEL
LIN {X 0,Y 665.682,Z 1158.041,A -85,B 0,C 180,E1 5286.989,E2 5286.989} C_VEL
LIN {X 0,Y 663.946,Z 1193.586,A -85,B 0,C 180,E1 5289.05,E2 5289.05} C_VEL
LIN {X 0,Y 662.254,Z 1226.914,A -85,B 0,C 180,E1 5291.663,E2 5291.663} C_VEL
LIN {X 0,Y 660.923,Z 1254.348,A -85,B 0,C 180,E1 5294.536,E2 5294.536} C_VEL
LIN {X 0,Y 660.136,Z 1276.508,A -85,B 0,C 180,E1 5297.615,E2 5297.615} C_VEL
LIN {X 0,Y 659.65,Z 1293.53,A -85,B 0,C 180,E1 5300.917,E2 5300.917} C_VEL
LIN {X 0,Y 659.509,Z 1304.515,A -85,B 0,C 180,E1 5304.072,E2 5304.072} C_VEL
LIN {X 0,Y 659.433,Z 1310.938,A -85,B 0,C 180,E1 5307.372,E2 5307.372} C_VEL
LIN {X 0,Y 659.384,Z 1312.5,A -85,B 0,C 180,E1 5310.006,E2 5310.006} C_VEL
LIN {X 0,Y 659.439,Z 1310.927,A -85,B 0,C 180,E1 5312.64,E2 5312.64} C_VEL
LIN {X 0,Y 659.523,Z 1304.476,A -85,B 0,C 180,E1 5315.94,E2 5315.94} C_VEL
LIN {X 0,Y 659.638,Z 1292.784,A -85,B 0,C 180,E1 5319.259,E2 5319.259} C_VEL
LIN {X 0,Y 660.151,Z 1276.439,A -85,B 0,C 180,E1 5322.395,E2 5322.395} C_VEL
LIN {X 0,Y 661.041,Z 1252.919,A -85,B 0,C 180,E1 5325.636,E2 5325.636} C_VEL
LIN {X 0,Y 662.201,Z 1227.058,A -85,B 0,C 180,E1 5328.325,E2 5328.325} C_VEL
LIN {X 0,Y 663.951,Z 1194.154,A -85,B 0,C 180,E1 5330.911,E2 5330.911} C_VEL
LIN {X 0,Y 665.656,Z 1158.849,A -85,B 0,C 180,E1 5332.971,E2 5332.971} C_VEL
LIN {X 0,Y 667.093,Z 1123.825,A -85,B 0,C 180,E1 5334.422,E2 5334.422} C_VEL
LIN {X 0,Y 668.149,Z 1082.286,A -85,B 0,C 180,E1 5335.531,E2 5335.531} C_VEL
LIN {X 0,Y 668.509,Z 1030.626,A -85,B 0,C 180,E1 5336.238,E2 5336.238} C_VEL
LIN {X 0,Y 669.048,Z 1022.207,A -85,B 0,C 180,E1 5336.396,E2 5336.396} C_VEL
LIN {X 0,Y 671.821,Z 1009.646,A -85,B 0,C 180,E1 5336.933,E2 5336.933} C_VEL
LIN {X 0,Y 663.805,Z 997.181,A -85,B 0,C 180,E1 5337.748,E2 5337.748} C_VEL
LIN {X 0,Y 658.788,Z 977.53,A -85,B 0,C 180,E1 5338.89,E2 5338.89} C_VEL
LIN {X 0,Y 658.72,Z 977.53,A -85,B 0,C 180,E1 5344.121,E2 5344.121} C_VEL
LIN {X 0,Y 658.656,Z 977.53,A -85,B 0,C 180,E1 5348.563,E2 5348.563} C_VEL
LIN {X 0,Y 658.745,Z 977.53,A -85,B 0,C 180,E1 5353.644,E2 5353.644} C_VEL
LIN {X 0,Y 658.604,Z 977.53,A -85,B 0,C 180,E1 5358.167,E2 5358.167} C_VEL
LIN {X 0,Y 658.661,Z 977.53,A -85,B 0,C 180,E1 5363.638,E2 5363.638} C_VEL
LIN {X 0,Y 658.737,Z 977.53,A -85,B 0,C 180,E1 5368.342,E2 5368.342} C_VEL
LIN {X 0,Y 658.856,Z 977.53,A -85,B 0,C 180,E1 5374.103,E2 5374.103} C_VEL
LIN {X 0,Y 658.907,Z 977.53,A -85,B 0,C 180,E1 5378.424,E2 5378.424} C_VEL
LIN {X 0,Y 658.959,Z 977.53,A -85,B 0,C 180,E1 5383.994,E2 5383.994} C_VEL
LIN {X 0,Y 659.041,Z 977.53,A -85,B 0,C 180,E1 5389.412,E2 5389.412} C_VEL
LIN {X 0,Y 659.139,Z 977.53,A -85,B 0,C 180,E1 5394.734,E2 5394.734} C_VEL
LIN {X 0,Y 659.197,Z 977.53,A -85,B 0,C 180,E1 5395.499,E2 5395.499} C_VEL
LIN {X 0,Y 663.087,Z 995.129,A -85,B 0,C 180,E1 5395.865,E2 5395.865} C_VEL
LIN {X 0,Y 662.665,Z 1051.117,A -85,B 0,C 180,E1 5396.692,E2 5396.692} C_VEL
LIN {X 0,Y 662.17,Z 1079.55,A -85,B 0,C 180,E1 5397.633,E2 5397.633} C_VEL
LIN {X 0,Y 661.492,Z 1104.988,A -85,B 0,C 180,E1 5399.025,E2 5399.025} C_VEL
LIN {X 0,Y 660.816,Z 1126.982,A -85,B 0,C 180,E1 5400.83,E2 5400.83} C_VEL
LIN {X 0,Y 660.289,Z 1144.974,A -85,B 0,C 180,E1 5403.03,E2 5403.03} C_VEL
LIN {X 0,Y 659.971,Z 1156.823,A -85,B 0,C 180,E1 5405.278,E2 5405.278} C_VEL
LIN {X 0,Y 659.774,Z 1163.06,A -85,B 0,C 180,E1 5407.265,E2 5407.265} C_VEL
LIN {X 0,Y 659.672,Z 1165.83,A -85,B 0,C 180,E1 5409.261,E2 5409.261} C_VEL
LIN {X 0,Y 659.717,Z 1164.239,A -85,B 0,C 180,E1 5411.938,E2 5411.938} C_VEL
LIN {X 0,Y 659.886,Z 1157.709,A -85,B 0,C 180,E1 5414.299,E2 5414.299} C_VEL
LIN {X 0,Y 660.171,Z 1145.524,A -85,B 0,C 180,E1 5416.681,E2 5416.681} C_VEL
LIN {X 0,Y 660.59,Z 1127.795,A -85,B 0,C 180,E1 5418.89,E2 5418.89} C_VEL
LIN {X 0,Y 661.185,Z 1105.836,A -85,B 0,C 180,E1 5420.727,E2 5420.727} C_VEL
LIN {X 0,Y 661.912,Z 1079.863,A -85,B 0,C 180,E1 5422.168,E2 5422.168} C_VEL
LIN {X 0,Y 662.375,Z 1051.759,A -85,B 0,C 180,E1 5423.124,E2 5423.124} C_VEL
LIN {X 0,Y 662.616,Z 1011.737,A -85,B 0,C 180,E1 5423.743,E2 5423.743} C_VEL
LIN {X 0,Y 661.981,Z 989.045,A -85,B 0,C 180,E1 5424.044,E2 5424.044} C_VEL
LIN {X 0,Y 659.106,Z 977.53,A -85,B 0,C 180,E1 5424.288,E2 5424.288} C_VEL
LIN {X 0,Y 658.73,Z 977.53,A -85,B 0,C 180,E1 5429.048,E2 5429.048} C_VEL
LIN {X 0,Y 658.667,Z 977.53,A -85,B 0,C 180,E1 5434.077,E2 5434.077} C_VEL
LIN {X 0,Y 658.676,Z 977.53,A -85,B 0,C 180,E1 5438.532,E2 5438.532} C_VEL
LIN {X 0,Y 658.759,Z 977.53,A -85,B 0,C 180,E1 5443.641,E2 5443.641} C_VEL
LIN {X 0,Y 658.589,Z 977.53,A -85,B 0,C 180,E1 5448.139,E2 5448.139} C_VEL
LIN {X 0,Y 658.642,Z 977.53,A -85,B 0,C 180,E1 5453.637,E2 5453.637} C_VEL
LIN {X 0,Y 658.782,Z 977.53,A -85,B 0,C 180,E1 5458.332,E2 5458.332} C_VEL
LIN {X 0,Y 658.846,Z 977.53,A -85,B 0,C 180,E1 5464.082,E2 5464.082} C_VEL
LIN {X 0,Y 658.892,Z 977.53,A -85,B 0,C 180,E1 5468.404,E2 5468.404} C_VEL
LIN {X 0,Y 658.983,Z 977.53,A -85,B 0,C 180,E1 5473.976,E2 5473.976} C_VEL
LIN {X 0,Y 659.072,Z 977.53,A -85,B 0,C 180,E1 5479.395,E2 5479.395} C_VEL
LIN {X 0,Y 659.128,Z 977.53,A -85,B 0,C 180,E1 5484.718,E2 5484.718} C_VEL
LIN {X 0,Y 659.228,Z 977.53,A -85,B 0,C 180,E1 5489.994,E2 5489.994} C_VEL
LIN {X 0,Y 659.287,Z 977.53,A -85,B 0,C 180,E1 5495.269,E2 5495.269} C_VEL
LIN {X 0,Y 658.987,Z 977.53,A -85,B 0,C 180,E1 5500.594,E2 5500.594} C_VEL
LIN {X 0,Y 658.985,Z 977.53,A -85,B 0,C 180,E1 5506.011,E2 5506.011} C_VEL
LIN {X 0,Y 658.868,Z 977.53,A -85,B 0,C 180,E1 5511.584,E2 5511.584} C_VEL
LIN {X 0,Y 658.806,Z 977.53,A -85,B 0,C 180,E1 5516.225,E2 5516.225} C_VEL
LIN {X 0,Y 658.757,Z 977.53,A -85,B 0,C 180,E1 5521.665,E2 5521.665} C_VEL
LIN {X 0,Y 658.741,Z 977.53,A -85,B 0,C 180,E1 5526.724,E2 5526.724} C_VEL
LIN {X 0,Y 658.713,Z 977.53,A -85,B 0,C 180,E1 5532.593,E2 5532.593} C_VEL
LIN {X 0,Y 658.631,Z 977.53,A -85,B 0,C 180,E1 5538.144,E2 5538.144} C_VEL
LIN {X 0,Y 658.671,Z 977.53,A -85,B 0,C 180,E1 5543.616,E2 5543.616} C_VEL
LIN {X 0,Y 658.756,Z 977.53,A -85,B 0,C 180,E1 5548.316,E2 5548.316} C_VEL
LIN {X 0,Y 658.942,Z 977.53,A -85,B 0,C 180,E1 5553.328,E2 5553.328} C_VEL
LIN {X 0,Y 668.624,Z 1005.598,A -85,B 0,C 180,E1 5554.07,E2 5554.07} C_VEL
LIN {X 0,Y 667.77,Z 1047.139,A -85,B 0,C 180,E1 5554.982,E2 5554.982} C_VEL
LIN {X 0,Y 666.307,Z 1085.51,A -85,B 0,C 180,E1 5556.364,E2 5556.364} C_VEL
LIN {X 0,Y 664.624,Z 1120.707,A -85,B 0,C 180,E1 5558.185,E2 5558.185} C_VEL
LIN {X 0,Y 662.985,Z 1153.362,A -85,B 0,C 180,E1 5560.465,E2 5560.465} C_VEL
LIN {X 0,Y 661.578,Z 1181.204,A -85,B 0,C 180,E1 5563.013,E2 5563.013} C_VEL
LIN {X 0,Y 660.544,Z 1205.19,A -85,B 0,C 180,E1 5565.885,E2 5565.885} C_VEL
LIN {X 0,Y 659.881,Z 1224.984,A -85,B 0,C 180,E1 5569.072,E2 5569.072} C_VEL
LIN {X 0,Y 659.605,Z 1239.469,A -85,B 0,C 180,E1 5572.401,E2 5572.401} C_VEL
LIN {X 0,Y 659.435,Z 1247.79,A -85,B 0,C 180,E1 5575.378,E2 5575.378} C_VEL
LIN {X 0,Y 659.367,Z 1252.112,A -85,B 0,C 180,E1 5578.674,E2 5578.674} C_VEL
LIN {X 0,Y 659.53,Z 1252.056,A -85,B 0,C 180,E1 5581.307,E2 5581.307} C_VEL
LIN {X 0,Y 659.477,Z 1247.639,A -85,B 0,C 180,E1 5584.603,E2 5584.603} C_VEL
LIN {X 0,Y 659.643,Z 1236.983,A -85,B 0,C 180,E1 5588.195,E2 5588.195} C_VEL
LIN {X 0,Y 660.051,Z 1220.948,A -85,B 0,C 180,E1 5591.577,E2 5591.577} C_VEL
LIN {X 0,Y 660.766,Z 1199.794,A -85,B 0,C 180,E1 5594.742,E2 5594.742} C_VEL
LIN {X 0,Y 661.868,Z 1174.688,A -85,B 0,C 180,E1 5597.555,E2 5597.555} C_VEL
LIN {X 0,Y 663.388,Z 1144.854,A -85,B 0,C 180,E1 5600.102,E2 5600.102} C_VEL
LIN {X 0,Y 664.992,Z 1111.969,A -85,B 0,C 180,E1 5602.232,E2 5602.232} C_VEL
LIN {X 0,Y 666.564,Z 1076.457,A -85,B 0,C 180,E1 5603.92,E2 5603.92} C_VEL
LIN {X 0,Y 665.884,Z 1068.65,A -85,B 0,C 180,E1 5604.254,E2 5604.254} C_VEL
LIN {X 0,Y 660.43,Z 1047.449,A -85,B 0,C 180,E1 5605.15,E2 5605.15} C_VEL
LIN {X 0,Y 660.36,Z 1045.368,A -85,B 0,C 180,E1 5605.21,E2 5605.21} C_VEL
LIN {X 0,Y 660.478,Z 1005.225,A -85,B 0,C 180,E1 5606.092,E2 5606.092} C_VEL
LIN {X 0,Y 650.824,Z 977.53,A -85,B 0,C 180,E1 5606.826,E2 5606.826} C_VEL
LIN {X 0,Y 650.797,Z 977.53,A -85,B 0,C 180,E1 5612.363,E2 5612.363} C_VEL
LIN {X 0,Y 650.712,Z 977.53,A -85,B 0,C 180,E1 5617.663,E2 5617.663} C_VEL
LIN {X 0,Y 650.595,Z 977.53,A -85,B 0,C 180,E1 5622.468,E2 5622.468} C_VEL
LIN {X 0,Y 650.616,Z 977.53,A -85,B 0,C 180,E1 5628.16,E2 5628.16} C_VEL
LIN {X 0,Y 650.773,Z 977.53,A -85,B 0,C 180,E1 5632.751,E2 5632.751} C_VEL
LIN {X 0,Y 650.765,Z 977.53,A -85,B 0,C 180,E1 5637.627,E2 5637.627} C_VEL
LIN {X 0,Y 650.805,Z 977.616,A -85,B 0,C 180,E1 5640.626,E2 5640.626} C_VEL
LIN {X 0,Y 657.92,Z 1003.125,A -85,B 0,C 180,E1 5642.214,E2 5642.214} C_VEL
LIN {X 0,Y 664.273,Z 1013.502,A -85,B 0,C 180,E1 5642.955,E2 5642.955} C_VEL
LIN {X 0,Y 661.565,Z 1024.025,A -85,B 0,C 180,E1 5643.403,E2 5643.403} C_VEL
LIN {X 0,Y 660.84,Z 1078.686,A -85,B 0,C 180,E1 5644.135,E2 5644.135} C_VEL
LIN {X 0,Y 659.64,Z 1120.921,A -85,B 0,C 180,E1 5645.259,E2 5645.259} C_VEL
LIN {X 0,Y 658.055,Z 1160.094,A -85,B 0,C 180,E1 5646.872,E2 5646.872} C_VEL
LIN {X 0,Y 656.436,Z 1193.892,A -85,B 0,C 180,E1 5648.821,E2 5648.821} C_VEL
LIN {X 0,Y 654.591,Z 1227.715,A -85,B 0,C 180,E1 5651.514,E2 5651.514} C_VEL
LIN {X 0,Y 653.157,Z 1255.109,A -85,B 0,C 180,E1 5654.443,E2 5654.443} C_VEL
LIN {X 0,Y 652.279,Z 1277.245,A -85,B 0,C 180,E1 5657.589,E2 5657.589} C_VEL
LIN {X 0,Y 651.757,Z 1294.218,A -85,B 0,C 180,E1 5660.971,E2 5660.971} C_VEL
LIN {X 0,Y 651.626,Z 1304.513,A -85,B 0,C 180,E1 5664,E2 5664} C_VEL
LIN {X 0,Y 651.529,Z 1310.933,A -85,B 0,C 180,E1 5667.34,E2 5667.34} C_VEL
LIN {X 0,Y 651.484,Z 1312.5,A -85,B 0,C 180,E1 5670.006,E2 5670.006} C_VEL
LIN {X 0,Y 651.535,Z 1310.925,A -85,B 0,C 180,E1 5672.672,E2 5672.672} C_VEL
LIN {X 0,Y 651.639,Z 1304.474,A -85,B 0,C 180,E1 5676.013,E2 5676.013} C_VEL
LIN {X 0,Y 651.77,Z 1292.779,A -85,B 0,C 180,E1 5679.372,E2 5679.372} C_VEL
LIN {X 0,Y 652.332,Z 1275.869,A -85,B 0,C 180,E1 5682.635,E2 5682.635} C_VEL
LIN {X 0,Y 653.362,Z 1251.852,A -85,B 0,C 180,E1 5685.956,E2 5685.956} C_VEL
LIN {X 0,Y 654.731,Z 1224.817,A -85,B 0,C 180,E1 5688.742,E2 5688.742} C_VEL
LIN {X 0,Y 656.591,Z 1192.326,A -85,B 0,C 180,E1 5691.282,E2 5691.282} C_VEL
LIN {X 0,Y 658.035,Z 1159.51,A -85,B 0,C 180,E1 5693.142,E2 5693.142} C_VEL
LIN {X 0,Y 659.542,Z 1121.33,A -85,B 0,C 180,E1 5694.686,E2 5694.686} C_VEL
LIN {X 0,Y 660.655,Z 1080.578,A -85,B 0,C 180,E1 5695.767,E2 5695.767} C_VEL
LIN {X 0,Y 661.034,Z 1028.121,A -85,B 0,C 180,E1 5696.486,E2 5696.486} C_VEL
LIN {X 0,Y 662.068,Z 1019.492,A -85,B 0,C 180,E1 5696.702,E2 5696.702} C_VEL
LIN {X 0,Y 663.325,Z 1011.749,A -85,B 0,C 180,E1 5697.048,E2 5697.048} C_VEL
LIN {X 0,Y 655.284,Z 996.934,A -85,B 0,C 180,E1 5697.993,E2 5697.993} C_VEL
LIN {X 0,Y 650.892,Z 977.53,A -85,B 0,C 180,E1 5699.141,E2 5699.141} C_VEL
LIN {X 0,Y 650.839,Z 977.53,A -85,B 0,C 180,E1 5703.978,E2 5703.978} C_VEL
LIN {X 0,Y 650.725,Z 977.53,A -85,B 0,C 180,E1 5708.963,E2 5708.963} C_VEL
LIN {X 0,Y 650.832,Z 977.53,A -85,B 0,C 180,E1 5714.312,E2 5714.312} C_VEL
LIN {X 0,Y 650.697,Z 977.53,A -85,B 0,C 180,E1 5719.324,E2 5719.324} C_VEL
LIN {X 0,Y 650.741,Z 977.53,A -85,B 0,C 180,E1 5724.596,E2 5724.596} C_VEL
LIN {X 0,Y 650.84,Z 977.53,A -85,B 0,C 180,E1 5729.489,E2 5729.489} C_VEL
LIN {X 0,Y 650.974,Z 977.53,A -85,B 0,C 180,E1 5733.766,E2 5733.766} C_VEL
LIN {X 0,Y 650.987,Z 977.53,A -85,B 0,C 180,E1 5738.617,E2 5738.617} C_VEL
LIN {X 0,Y 651.037,Z 977.53,A -85,B 0,C 180,E1 5743.794,E2 5743.794} C_VEL
LIN {X 0,Y 651.116,Z 977.53,A -85,B 0,C 180,E1 5749.281,E2 5749.281} C_VEL
LIN {X 0,Y 651.263,Z 977.53,A -85,B 0,C 180,E1 5754.67,E2 5754.67} C_VEL
LIN {X 0,Y 651.278,Z 977.53,A -85,B 0,C 180,E1 5755.246,E2 5755.246} C_VEL
LIN {X 0,Y 655.634,Z 995.358,A -85,B 0,C 180,E1 5755.646,E2 5755.646} C_VEL
LIN {X 0,Y 655.1,Z 1052.889,A -85,B 0,C 180,E1 5756.529,E2 5756.529} C_VEL
LIN {X 0,Y 654.594,Z 1079.914,A -85,B 0,C 180,E1 5757.439,E2 5757.439} C_VEL
LIN {X 0,Y 653.852,Z 1105.542,A -85,B 0,C 180,E1 5758.848,E2 5758.848} C_VEL
LIN {X 0,Y 653.114,Z 1127.612,A -85,B 0,C 180,E1 5760.674,E2 5760.674} C_VEL
LIN {X 0,Y 652.536,Z 1145.335,A -85,B 0,C 180,E1 5762.841,E2 5762.841} C_VEL
LIN {X 0,Y 652.179,Z 1158.3,A -85,B 0,C 180,E1 5765.341,E2 5765.341} C_VEL
LIN {X 0,Y 651.861,Z 1165.526,A -85,B 0,C 180,E1 5768.026,E2 5768.026} C_VEL
LIN {X 0,Y 651.857,Z 1166.64,A -85,B 0,C 180,E1 5770.726,E2 5770.726} C_VEL
LIN {X 0,Y 651.989,Z 1161.672,A -85,B 0,C 180,E1 5773.447,E2 5773.447} C_VEL
LIN {X 0,Y 652.216,Z 1151.718,A -85,B 0,C 180,E1 5775.86,E2 5775.86} C_VEL
LIN {X 0,Y 652.657,Z 1136.155,A -85,B 0,C 180,E1 5778.168,E2 5778.168} C_VEL
LIN {X 0,Y 653.271,Z 1115.656,A -85,B 0,C 180,E1 5780.183,E2 5780.183} C_VEL
LIN {X 0,Y 653.97,Z 1091.907,A -85,B 0,C 180,E1 5781.768,E2 5781.768} C_VEL
LIN {X 0,Y 654.575,Z 1063.897,A -85,B 0,C 180,E1 5782.967,E2 5782.967} C_VEL
LIN {X 0,Y 654.904,Z 1033.095,A -85,B 0,C 180,E1 5783.663,E2 5783.663} C_VEL
LIN {X 0,Y 654.252,Z 989.824,A -85,B 0,C 180,E1 5784.23,E2 5784.23} C_VEL
LIN {X 0,Y 651.139,Z 977.53,A -85,B 0,C 180,E1 5784.515,E2 5784.515} C_VEL
LIN {X 0,Y 650.857,Z 977.53,A -85,B 0,C 180,E1 5790.514,E2 5790.514} C_VEL
LIN {X 0,Y 650.775,Z 977.53,A -85,B 0,C 180,E1 5795.605,E2 5795.605} C_VEL
LIN {X 0,Y 650.751,Z 977.53,A -85,B 0,C 180,E1 5800.697,E2 5800.697} C_VEL
LIN {X 0,Y 650.795,Z 977.53,A -85,B 0,C 180,E1 5805.685,E2 5805.685} C_VEL
LIN {X 0,Y 650.672,Z 977.53,A -85,B 0,C 180,E1 5811.033,E2 5811.033} C_VEL
LIN {X 0,Y 650.734,Z 977.53,A -85,B 0,C 180,E1 5816.016,E2 5816.016} C_VEL
LIN {X 0,Y 650.833,Z 977.53,A -85,B 0,C 180,E1 5820.723,E2 5820.723} C_VEL
LIN {X 0,Y 650.945,Z 977.53,A -85,B 0,C 180,E1 5825.222,E2 5825.222} C_VEL
LIN {X 0,Y 650.972,Z 977.53,A -85,B 0,C 180,E1 5829.558,E2 5829.558} C_VEL
LIN {X 0,Y 651.058,Z 977.53,A -85,B 0,C 180,E1 5833.776,E2 5833.776} C_VEL
LIN {X 0,Y 651.149,Z 977.53,A -85,B 0,C 180,E1 5839.265,E2 5839.265} C_VEL
LIN {X 0,Y 651.252,Z 977.53,A -85,B 0,C 180,E1 5844.654,E2 5844.654} C_VEL
LIN {X 0,Y 651.336,Z 977.53,A -85,B 0,C 180,E1 5849.994,E2 5849.994} C_VEL
LIN {X 0,Y 651.381,Z 977.53,A -85,B 0,C 180,E1 5855.333,E2 5855.333} C_VEL
LIN {X 0,Y 651.077,Z 977.53,A -85,B 0,C 180,E1 5860.724,E2 5860.724} C_VEL
LIN {X 0,Y 651.064,Z 977.53,A -85,B 0,C 180,E1 5866.211,E2 5866.211} C_VEL
LIN {X 0,Y 650.956,Z 977.53,A -85,B 0,C 180,E1 5871.384,E2 5871.384} C_VEL
LIN {X 0,Y 650.926,Z 977.53,A -85,B 0,C 180,E1 5876.243,E2 5876.243} C_VEL
LIN {X 0,Y 650.829,Z 977.53,A -85,B 0,C 180,E1 5880.804,E2 5880.804} C_VEL
LIN {X 0,Y 650.814,Z 977.53,A -85,B 0,C 180,E1 5885.588,E2 5885.588} C_VEL
LIN {X 0,Y 650.766,Z 977.53,A -85,B 0,C 180,E1 5890.681,E2 5890.681} C_VEL
LIN {X 0,Y 650.775,Z 977.53,A -85,B 0,C 180,E1 5895.685,E2 5895.685} C_VEL
LIN {X 0,Y 650.675,Z 977.53,A -85,B 0,C 180,E1 5901.034,E2 5901.034} C_VEL
LIN {X 0,Y 650.728,Z 977.53,A -85,B 0,C 180,E1 5906.016,E2 5906.016} C_VEL
LIN {X 0,Y 650.855,Z 977.53,A -85,B 0,C 180,E1 5910.724,E2 5910.724} C_VEL
LIN {X 0,Y 651.007,Z 977.53,A -85,B 0,C 180,E1 5913.01,E2 5913.01} C_VEL
LIN {X 0,Y 661.361,Z 1008.313,A -85,B 0,C 180,E1 5913.835,E2 5913.835} C_VEL
LIN {X 0,Y 660.398,Z 1049.839,A -85,B 0,C 180,E1 5914.798,E2 5914.798} C_VEL
LIN {X 0,Y 658.847,Z 1086.915,A -85,B 0,C 180,E1 5916.17,E2 5916.17} C_VEL
LIN {X 0,Y 657.087,Z 1122.191,A -85,B 0,C 180,E1 5918.023,E2 5918.023} C_VEL
LIN {X 0,Y 655.342,Z 1154.396,A -85,B 0,C 180,E1 5920.316,E2 5920.316} C_VEL
LIN {X 0,Y 653.8,Z 1182.787,A -85,B 0,C 180,E1 5922.978,E2 5922.978} C_VEL
LIN {X 0,Y 652.716,Z 1206.38,A -85,B 0,C 180,E1 5925.884,E2 5925.884} C_VEL
LIN {X 0,Y 652.044,Z 1224.98,A -85,B 0,C 180,E1 5928.939,E2 5928.939} C_VEL
LIN {X 0,Y 651.74,Z 1239.467,A -85,B 0,C 180,E1 5932.309,E2 5932.309} C_VEL
LIN {X 0,Y 651.546,Z 1247.789,A -85,B 0,C 180,E1 5935.322,E2 5935.322} C_VEL
LIN {X 0,Y 651.469,Z 1252.111,A -85,B 0,C 180,E1 5938.658,E2 5938.658} C_VEL
LIN {X 0,Y 651.629,Z 1252.057,A -85,B 0,C 180,E1 5941.323,E2 5941.323} C_VEL
LIN {X 0,Y 651.584,Z 1247.64,A -85,B 0,C 180,E1 5944.659,E2 5944.659} C_VEL
LIN {X 0,Y 651.717,Z 1238.084,A -85,B 0,C 180,E1 5948.008,E2 5948.008} C_VEL
LIN {X 0,Y 652.177,Z 1222.876,A -85,B 0,C 180,E1 5951.379,E2 5951.379} C_VEL
LIN {X 0,Y 652.888,Z 1202.219,A -85,B 0,C 180,E1 5954.608,E2 5954.608} C_VEL
LIN {X 0,Y 654.125,Z 1176.175,A -85,B 0,C 180,E1 5957.621,E2 5957.621} C_VEL
LIN {X 0,Y 655.722,Z 1147.015,A -85,B 0,C 180,E1 5960.18,E2 5960.18} C_VEL
LIN {X 0,Y 657.362,Z 1115.5,A -85,B 0,C 180,E1 5962.282,E2 5962.282} C_VEL
LIN {X 0,Y 659.042,Z 1079.787,A -85,B 0,C 180,E1 5964.028,E2 5964.028} C_VEL
LIN {X 0,Y 660.36,Z 1045.368,A -85,B 0,C 180,E1 5965.21,E2 5965.21} C_VEL
LIN {X 0,Y 657.121,Z 1029.237,A -85,B 0,C 180,E1 5965.742,E2 5965.742} C_VEL
LIN {X 0,Y 653.835,Z 1012.891,A -85,B 0,C 180,E1 5966.197,E2 5966.197} C_VEL
LIN {X 0,Y 652.186,Z 1004.66,A -85,B 0,C 180,E1 5966.389,E2 5966.389} C_VEL
LIN {X 0,Y 642.921,Z 977.53,A -85,B 0,C 180,E1 5967.108,E2 5967.108} C_VEL
LIN {X 0,Y 642.891,Z 977.53,A -85,B 0,C 180,E1 5972.811,E2 5972.811} C_VEL
LIN {X 0,Y 642.795,Z 977.53,A -85,B 0,C 180,E1 5977.782,E2 5977.782} C_VEL
LIN {X 0,Y 642.647,Z 977.53,A -85,B 0,C 180,E1 5983.12,E2 5983.12} C_VEL
LIN {X 0,Y 642.708,Z 977.53,A -85,B 0,C 180,E1 5988.954,E2 5988.954} C_VEL
LIN {X 0,Y 642.877,Z 977.53,A -85,B 0,C 180,E1 5993.904,E2 5993.904} C_VEL
LIN {X 0,Y 642.816,Z 977.53,A -85,B 0,C 180,E1 5998.77,E2 5998.77} C_VEL
LIN {X 0,Y 642.907,Z 977.941,A -85,B 0,C 180,E1 6000.341,E2 6000.341} C_VEL
LIN {X 0,Y 650.177,Z 1005.016,A -85,B 0,C 180,E1 6002.049,E2 6002.049} C_VEL
LIN {X 0,Y 655.865,Z 1016.958,A -85,B 0,C 180,E1 6002.859,E2 6002.859} C_VEL
LIN {X 0,Y 654.196,Z 1026.326,A -85,B 0,C 180,E1 6003.168,E2 6003.168} C_VEL
LIN {X 0,Y 653.44,Z 1079.267,A -85,B 0,C 180,E1 6003.904,E2 6003.904} C_VEL
LIN {X 0,Y 652.109,Z 1121.254,A -85,B 0,C 180,E1 6005.052,E2 6005.052} C_VEL
LIN {X 0,Y 650.452,Z 1159.987,A -85,B 0,C 180,E1 6006.677,E2 6006.677} C_VEL
LIN {X 0,Y 648.615,Z 1196.675,A -85,B 0,C 180,E1 6008.825,E2 6008.825} C_VEL
LIN {X 0,Y 647.027,Z 1226.691,A -85,B 0,C 180,E1 6011.197,E2 6011.197} C_VEL
LIN {X 0,Y 645.528,Z 1253.042,A -85,B 0,C 180,E1 6013.996,E2 6013.996} C_VEL
LIN {X 0,Y 644.497,Z 1276.193,A -85,B 0,C 180,E1 6017.259,E2 6017.259} C_VEL
LIN {X 0,Y 643.932,Z 1292.823,A -85,B 0,C 180,E1 6020.525,E2 6020.525} C_VEL
LIN {X 0,Y 643.754,Z 1304.511,A -85,B 0,C 180,E1 6023.926,E2 6023.926} C_VEL
LIN {X 0,Y 643.625,Z 1310.928,A -85,B 0,C 180,E1 6027.307,E2 6027.307} C_VEL
LIN {X 0,Y 643.611,Z 1312.5,A -85,B 0,C 180,E1 6030.006,E2 6030.006} C_VEL
LIN {X 0,Y 643.631,Z 1310.921,A -85,B 0,C 180,E1 6032.705,E2 6032.705} C_VEL
LIN {X 0,Y 643.767,Z 1304.472,A -85,B 0,C 180,E1 6036.086,E2 6036.086} C_VEL
LIN {X 0,Y 643.901,Z 1292.773,A -85,B 0,C 180,E1 6039.488,E2 6039.488} C_VEL
LIN {X 0,Y 644.529,Z 1276.096,A -85,B 0,C 180,E1 6042.754,E2 6042.754} C_VEL
LIN {X 0,Y 645.568,Z 1252.934,A -85,B 0,C 180,E1 6046.017,E2 6046.017} C_VEL
LIN {X 0,Y 647.03,Z 1226.688,A -85,B 0,C 180,E1 6048.803,E2 6048.803} C_VEL
LIN {X 0,Y 648.566,Z 1198.338,A -85,B 0,C 180,E1 6051.045,E2 6051.045} C_VEL
LIN {X 0,Y 650.232,Z 1162.714,A -85,B 0,C 180,E1 6053.137,E2 6053.137} C_VEL
LIN {X 0,Y 651.84,Z 1123.615,A -85,B 0,C 180,E1 6054.789,E2 6054.789} C_VEL
LIN {X 0,Y 653.058,Z 1082.966,A -85,B 0,C 180,E1 6055.923,E2 6055.923} C_VEL
LIN {X 0,Y 653.547,Z 1035.89,A -85,B 0,C 180,E1 6056.622,E2 6056.622} C_VEL
LIN {X 0,Y 654.077,Z 1021.185,A -85,B 0,C 180,E1 6056.822,E2 6056.822} C_VEL
LIN {X 0,Y 655.54,Z 1015.27,A -85,B 0,C 180,E1 6057.077,E2 6057.077} C_VEL
LIN {X 0,Y 646.542,Z 995.759,A -85,B 0,C 180,E1 6058.3,E2 6058.3} C_VEL
LIN {X 0,Y 642.969,Z 977.53,A -85,B 0,C 180,E1 6059.344,E2 6059.344} C_VEL
LIN {X 0,Y 642.909,Z 977.53,A -85,B 0,C 180,E1 6064.455,E2 6064.455} C_VEL
LIN {X 0,Y 642.829,Z 977.53,A -85,B 0,C 180,E1 6069.535,E2 6069.535} C_VEL
LIN {X 0,Y 642.879,Z 977.53,A -85,B 0,C 180,E1 6075.021,E2 6075.021} C_VEL
LIN {X 0,Y 642.763,Z 977.53,A -85,B 0,C 180,E1 6080.486,E2 6080.486} C_VEL
LIN {X 0,Y 642.807,Z 977.53,A -85,B 0,C 180,E1 6085.604,E2 6085.604} C_VEL
LIN {X 0,Y 642.971,Z 977.53,A -85,B 0,C 180,E1 6090.7,E2 6090.7} C_VEL
LIN {X 0,Y 643.055,Z 977.53,A -85,B 0,C 180,E1 6094.917,E2 6094.917} C_VEL
LIN {X 0,Y 643.074,Z 977.53,A -85,B 0,C 180,E1 6100.496,E2 6100.496} C_VEL
LIN {X 0,Y 643.107,Z 977.53,A -85,B 0,C 180,E1 6105.046,E2 6105.046} C_VEL
LIN {X 0,Y 643.253,Z 977.53,A -85,B 0,C 180,E1 6110.52,E2 6110.52} C_VEL
LIN {X 0,Y 643.426,Z 978.295,A -85,B 0,C 180,E1 6114.997,E2 6114.997} C_VEL
LIN {X 0,Y 648.153,Z 997.914,A -85,B 0,C 180,E1 6115.451,E2 6115.451} C_VEL
LIN {X 0,Y 647.529,Z 1054.709,A -85,B 0,C 180,E1 6116.362,E2 6116.362} C_VEL
LIN {X 0,Y 646.943,Z 1082.259,A -85,B 0,C 180,E1 6117.325,E2 6117.325} C_VEL
LIN {X 0,Y 646.207,Z 1107.289,A -85,B 0,C 180,E1 6118.75,E2 6118.75} C_VEL
LIN {X 0,Y 645.377,Z 1129.92,A -85,B 0,C 180,E1 6120.682,E2 6120.682} C_VEL
LIN {X 0,Y 644.773,Z 1147.172,A -85,B 0,C 180,E1 6122.876,E2 6122.876} C_VEL
LIN {X 0,Y 644.347,Z 1159.748,A -85,B 0,C 180,E1 6125.407,E2 6125.407} C_VEL
LIN {X 0,Y 644.027,Z 1166.679,A -85,B 0,C 180,E1 6128.124,E2 6128.124} C_VEL
LIN {X 0,Y 644.039,Z 1167.468,A -85,B 0,C 180,E1 6130.857,E2 6130.857} C_VEL
LIN {X 0,Y 644.167,Z 1162.224,A -85,B 0,C 180,E1 6133.613,E2 6133.613} C_VEL
LIN {X 0,Y 644.463,Z 1151.829,A -85,B 0,C 180,E1 6136.079,E2 6136.079} C_VEL
LIN {X 0,Y 644.939,Z 1135.056,A -85,B 0,C 180,E1 6138.5,E2 6138.5} C_VEL
LIN {X 0,Y 645.681,Z 1113.666,A -85,B 0,C 180,E1 6140.538,E2 6140.538} C_VEL
LIN {X 0,Y 646.389,Z 1088.665,A -85,B 0,C 180,E1 6142.132,E2 6142.132} C_VEL
LIN {X 0,Y 647.066,Z 1059.945,A -85,B 0,C 180,E1 6143.284,E2 6143.284} C_VEL
LIN {X 0,Y 647.365,Z 1029.32,A -85,B 0,C 180,E1 6143.902,E2 6143.902} C_VEL
LIN {X 0,Y 646.834,Z 991.814,A -85,B 0,C 180,E1 6144.398,E2 6144.398} C_VEL
LIN {X 0,Y 643.193,Z 977.53,A -85,B 0,C 180,E1 6144.716,E2 6144.716} C_VEL
LIN {X 0,Y 642.905,Z 977.53,A -85,B 0,C 180,E1 6149.674,E2 6149.674} C_VEL
LIN {X 0,Y 642.865,Z 977.53,A -85,B 0,C 180,E1 6154.457,E2 6154.457} C_VEL
LIN {X 0,Y 642.831,Z 977.53,A -85,B 0,C 180,E1 6159.533,E2 6159.533} C_VEL
LIN {X 0,Y 642.872,Z 977.53,A -85,B 0,C 180,E1 6165.007,E2 6165.007} C_VEL
LIN {X 0,Y 642.762,Z 977.53,A -85,B 0,C 180,E1 6170.46,E2 6170.46} C_VEL
LIN {X 0,Y 642.799,Z 977.53,A -85,B 0,C 180,E1 6175.601,E2 6175.601} C_VEL
LIN {X 0,Y 642.962,Z 977.53,A -85,B 0,C 180,E1 6180.697,E2 6180.697} C_VEL
LIN {X 0,Y 643.052,Z 977.53,A -85,B 0,C 180,E1 6184.897,E2 6184.897} C_VEL
LIN {X 0,Y 643.048,Z 977.53,A -85,B 0,C 180,E1 6190.494,E2 6190.494} C_VEL
LIN {X 0,Y 643.151,Z 977.53,A -85,B 0,C 180,E1 6195.02,E2 6195.02} C_VEL
LIN {X 0,Y 643.264,Z 977.53,A -85,B 0,C 180,E1 6200.503,E2 6200.503} C_VEL
LIN {X 0,Y 643.416,Z 977.53,A -85,B 0,C 180,E1 6205.942,E2 6205.942} C_VEL
LIN {X 0,Y 643.583,Z 977.53,A -85,B 0,C 180,E1 6211.343,E2 6211.343} C_VEL
LIN {X 0,Y 643.239,Z 977.53,A -85,B 0,C 180,E1 6216.758,E2 6216.758} C_VEL
LIN {X 0,Y 643.224,Z 977.53,A -85,B 0,C 180,E1 6222.234,E2 6222.234} C_VEL
LIN {X 0,Y 643.142,Z 977.53,A -85,B 0,C 180,E1 6227.829,E2 6227.829} C_VEL
LIN {X 0,Y 643.016,Z 977.53,A -85,B 0,C 180,E1 6233.206,E2 6233.206} C_VEL
LIN {X 0,Y 642.95,Z 977.53,A -85,B 0,C 180,E1 6238.115,E2 6238.115} C_VEL
LIN {X 0,Y 642.892,Z 977.53,A -85,B 0,C 180,E1 6242.819,E2 6242.819} C_VEL
LIN {X 0,Y 642.827,Z 977.53,A -85,B 0,C 180,E1 6247.789,E2 6247.789} C_VEL
LIN {X 0,Y 642.885,Z 977.53,A -85,B 0,C 180,E1 6253.111,E2 6253.111} C_VEL
LIN {X 0,Y 642.816,Z 977.53,A -85,B 0,C 180,E1 6258.956,E2 6258.956} C_VEL
LIN {X 0,Y 642.771,Z 977.53,A -85,B 0,C 180,E1 6263.882,E2 6263.882} C_VEL
LIN {X 0,Y 642.854,Z 977.53,A -85,B 0,C 180,E1 6268.757,E2 6268.757} C_VEL
LIN {X 0,Y 643.082,Z 977.53,A -85,B 0,C 180,E1 6272.685,E2 6272.685} C_VEL
LIN {X 0,Y 654.112,Z 1009.329,A -85,B 0,C 180,E1 6273.57,E2 6273.57} C_VEL
LIN {X 0,Y 653.046,Z 1051.393,A -85,B 0,C 180,E1 6274.574,E2 6274.574} C_VEL
LIN {X 0,Y 651.417,Z 1088.321,A -85,B 0,C 180,E1 6275.972,E2 6275.972} C_VEL
LIN {X 0,Y 649.533,Z 1123.627,A -85,B 0,C 180,E1 6277.866,E2 6277.866} C_VEL
LIN {X 0,Y 647.698,Z 1155.398,A -85,B 0,C 180,E1 6280.163,E2 6280.163} C_VEL
LIN {X 0,Y 646.097,Z 1182.779,A -85,B 0,C 180,E1 6282.769,E2 6282.769} C_VEL
LIN {X 0,Y 644.934,Z 1206.374,A -85,B 0,C 180,E1 6285.71,E2 6285.71} C_VEL
LIN {X 0,Y 644.21,Z 1224.976,A -85,B 0,C 180,E1 6288.802,E2 6288.802} C_VEL
LIN {X 0,Y 643.867,Z 1239.465,A -85,B 0,C 180,E1 6292.214,E2 6292.214} C_VEL
LIN {X 0,Y 643.649,Z 1247.788,A -85,B 0,C 180,E1 6295.265,E2 6295.265} C_VEL
LIN {X 0,Y 643.568,Z 1252.111,A -85,B 0,C 180,E1 6298.641,E2 6298.641} C_VEL
LIN {X 0,Y 643.727,Z 1252.057,A -85,B 0,C 180,E1 6301.339,E2 6301.339} C_VEL
LIN {X 0,Y 643.691,Z 1247.641,A -85,B 0,C 180,E1 6304.716,E2 6304.716} C_VEL
LIN {X 0,Y 643.834,Z 1238.086,A -85,B 0,C 180,E1 6308.107,E2 6308.107} C_VEL
LIN {X 0,Y 644.317,Z 1222.879,A -85,B 0,C 180,E1 6311.52,E2 6311.52} C_VEL
LIN {X 0,Y 645.121,Z 1202.221,A -85,B 0,C 180,E1 6314.787,E2 6314.787} C_VEL
LIN {X 0,Y 646.398,Z 1177.244,A -85,B 0,C 180,E1 6317.73,E2 6317.73} C_VEL
LIN {X 0,Y 648.099,Z 1148.029,A -85,B 0,C 180,E1 6320.339,E2 6320.339} C_VEL
LIN {X 0,Y 649.894,Z 1114.989,A -85,B 0,C 180,E1 6322.551,E2 6322.551} C_VEL
LIN {X 0,Y 651.654,Z 1078.753,A -85,B 0,C 180,E1 6324.317,E2 6324.317} C_VEL
LIN {X 0,Y 653.063,Z 1040.951,A -85,B 0,C 180,E1 6325.583,E2 6325.583} C_VEL
LIN {X 0,Y 653.835,Z 1012.891,A -85,B 0,C 180,E1 6326.197,E2 6326.197} C_VEL
LIN {X 0,Y 651.233,Z 1006.716,A -85,B 0,C 180,E1 6326.399,E2 6326.399} C_VEL
LIN {X 0,Y 641.14,Z 996.544,A -85,B 0,C 180,E1 6326.906,E2 6326.906} C_VEL
LIN {X 0,Y 640.524,Z 995.199,A -85,B 0,C 180,E1 6326.945,E2 6326.945} C_VEL
LIN {X 0,Y 635.015,Z 977.53,A -85,B 0,C 180,E1 6327.406,E2 6327.406} C_VEL
LIN {X 0,Y 634.938,Z 977.53,A -85,B 0,C 180,E1 6333.275,E2 6333.275} C_VEL
LIN {X 0,Y 634.893,Z 977.53,A -85,B 0,C 180,E1 6338.337,E2 6338.337} C_VEL
LIN {X 0,Y 634.652,Z 977.53,A -85,B 0,C 180,E1 6344.262,E2 6344.262} C_VEL
LIN {X 0,Y 634.787,Z 977.53,A -85,B 0,C 180,E1 6349.88,E2 6349.88} C_VEL
LIN {X 0,Y 634.98,Z 977.53,A -85,B 0,C 180,E1 6355.068,E2 6355.068} C_VEL
LIN {X 0,Y 634.997,Z 977.805,A -85,B 0,C 180,E1 6360.023,E2 6360.023} C_VEL
LIN {X 0,Y 643.14,Z 1008.465,A -85,B 0,C 180,E1 6361.985,E2 6361.985} C_VEL
LIN {X 0,Y 648.117,Z 1017.706,A -85,B 0,C 180,E1 6362.641,E2 6362.641} C_VEL
LIN {X 0,Y 646.998,Z 1024.031,A -85,B 0,C 180,E1 6362.879,E2 6362.879} C_VEL
LIN {X 0,Y 646.066,Z 1078.337,A -85,B 0,C 180,E1 6363.638,E2 6363.638} C_VEL
LIN {X 0,Y 644.715,Z 1118.94,A -85,B 0,C 180,E1 6364.746,E2 6364.746} C_VEL
LIN {X 0,Y 642.93,Z 1158.139,A -85,B 0,C 180,E1 6366.388,E2 6366.388} C_VEL
LIN {X 0,Y 641.051,Z 1194.46,A -85,B 0,C 180,E1 6368.515,E2 6368.515} C_VEL
LIN {X 0,Y 639.212,Z 1227.563,A -85,B 0,C 180,E1 6371.121,E2 6371.121} C_VEL
LIN {X 0,Y 637.827,Z 1253.031,A -85,B 0,C 180,E1 6373.797,E2 6373.797} C_VEL
LIN {X 0,Y 636.671,Z 1276.492,A -85,B 0,C 180,E1 6377.149,E2 6377.149} C_VEL
LIN {X 0,Y 636.064,Z 1292.817,A -85,B 0,C 180,E1 6380.407,E2 6380.407} C_VEL
LIN {X 0,Y 635.861,Z 1304.51,A -85,B 0,C 180,E1 6383.85,E2 6383.85} C_VEL
LIN {X 0,Y 635.737,Z 1310.923,A -85,B 0,C 180,E1 6387.274,E2 6387.274} C_VEL
LIN {X 0,Y 635.726,Z 1312.5,A -85,B 0,C 180,E1 6390.006,E2 6390.006} C_VEL
LIN {X 0,Y 635.743,Z 1310.915,A -85,B 0,C 180,E1 6392.739,E2 6392.739} C_VEL
LIN {X 0,Y 635.874,Z 1304.47,A -85,B 0,C 180,E1 6396.162,E2 6396.162} C_VEL
LIN {X 0,Y 636.033,Z 1292.767,A -85,B 0,C 180,E1 6399.606,E2 6399.606} C_VEL
LIN {X 0,Y 636.715,Z 1276.614,A -85,B 0,C 180,E1 6402.83,E2 6402.83} C_VEL
LIN {X 0,Y 637.866,Z 1252.924,A -85,B 0,C 180,E1 6406.216,E2 6406.216} C_VEL
LIN {X 0,Y 639.138,Z 1228.778,A -85,B 0,C 180,E1 6408.754,E2 6408.754} C_VEL
LIN {X 0,Y 640.863,Z 1196.436,A -85,B 0,C 180,E1 6411.299,E2 6411.299} C_VEL
LIN {X 0,Y 642.565,Z 1161.155,A -85,B 0,C 180,E1 6413.376,E2 6413.376} C_VEL
LIN {X 0,Y 644.332,Z 1120.497,A -85,B 0,C 180,E1 6415.098,E2 6415.098} C_VEL
LIN {X 0,Y 645.702,Z 1081.034,A -85,B 0,C 180,E1 6416.205,E2 6416.205} C_VEL
LIN {X 0,Y 646.323,Z 1028.379,A -85,B 0,C 180,E1 6416.976,E2 6416.976} C_VEL
LIN {X 0,Y 647.384,Z 1017.476,A -85,B 0,C 180,E1 6417.183,E2 6417.183} C_VEL
LIN {X 0,Y 638.327,Z 994.805,A -85,B 0,C 180,E1 6418.594,E2 6418.594} C_VEL
LIN {X 0,Y 635.035,Z 977.53,A -85,B 0,C 180,E1 6419.626,E2 6419.626} C_VEL
LIN {X 0,Y 634.934,Z 977.53,A -85,B 0,C 180,E1 6424.95,E2 6424.95} C_VEL
LIN {X 0,Y 634.875,Z 977.53,A -85,B 0,C 180,E1 6430.227,E2 6430.227} C_VEL
LIN {X 0,Y 634.898,Z 977.53,A -85,B 0,C 180,E1 6435.733,E2 6435.733} C_VEL
LIN {X 0,Y 634.854,Z 977.53,A -85,B 0,C 180,E1 6441.66,E2 6441.66} C_VEL
LIN {X 0,Y 634.872,Z 977.53,A -85,B 0,C 180,E1 6446.721,E2 6446.721} C_VEL
LIN {X 0,Y 635.077,Z 977.53,A -85,B 0,C 180,E1 6451.996,E2 6451.996} C_VEL
LIN {X 0,Y 635.139,Z 977.53,A -85,B 0,C 180,E1 6457.573,E2 6457.573} C_VEL
LIN {X 0,Y 635.196,Z 977.53,A -85,B 0,C 180,E1 6462.613,E2 6462.613} C_VEL
LIN {X 0,Y 635.241,Z 977.53,A -85,B 0,C 180,E1 6467.986,E2 6467.986} C_VEL
LIN {X 0,Y 635.479,Z 977.53,A -85,B 0,C 180,E1 6473.163,E2 6473.163} C_VEL
LIN {X 0,Y 635.494,Z 977.53,A -85,B 0,C 180,E1 6474.697,E2 6474.697} C_VEL
LIN {X 0,Y 640.73,Z 998.21,A -85,B 0,C 180,E1 6475.215,E2 6475.215} C_VEL
LIN {X 0,Y 640.016,Z 1054.982,A -85,B 0,C 180,E1 6476.15,E2 6476.15} C_VEL
LIN {X 0,Y 639.388,Z 1082.663,A -85,B 0,C 180,E1 6477.123,E2 6477.123} C_VEL
LIN {X 0,Y 638.578,Z 1107.88,A -85,B 0,C 180,E1 6478.565,E2 6478.565} C_VEL
LIN {X 0,Y 637.684,Z 1130.576,A -85,B 0,C 180,E1 6480.52,E2 6480.52} C_VEL
LIN {X 0,Y 637.025,Z 1147.903,A -85,B 0,C 180,E1 6482.736,E2 6482.736} C_VEL
LIN {X 0,Y 636.574,Z 1159.95,A -85,B 0,C 180,E1 6485.13,E2 6485.13} C_VEL
LIN {X 0,Y 636.262,Z 1166.736,A -85,B 0,C 180,E1 6487.535,E2 6487.535} C_VEL
LIN {X 0,Y 636.174,Z 1168.779,A -85,B 0,C 180,E1 6489.606,E2 6489.606} C_VEL
LIN {X 0,Y 636.265,Z 1166.213,A -85,B 0,C 180,E1 6492.44,E2 6492.44} C_VEL
LIN {X 0,Y 636.495,Z 1158.925,A -85,B 0,C 180,E1 6494.836,E2 6494.836} C_VEL
LIN {X 0,Y 636.886,Z 1146.122,A -85,B 0,C 180,E1 6497.25,E2 6497.25} C_VEL
LIN {X 0,Y 637.477,Z 1128.179,A -85,B 0,C 180,E1 6499.445,E2 6499.445} C_VEL
LIN {X 0,Y 638.227,Z 1105.646,A -85,B 0,C 180,E1 6501.318,E2 6501.318} C_VEL
LIN {X 0,Y 639.078,Z 1079.509,A -85,B 0,C 180,E1 6502.761,E2 6502.761} C_VEL
LIN {X 0,Y 639.642,Z 1051.153,A -85,B 0,C 180,E1 6503.709,E2 6503.709} C_VEL
LIN {X 0,Y 639.234,Z 993.035,A -85,B 0,C 180,E1 6504.589,E2 6504.589} C_VEL
LIN {X 0,Y 635.265,Z 977.53,A -85,B 0,C 180,E1 6504.974,E2 6504.974} C_VEL
LIN {X 0,Y 634.948,Z 977.53,A -85,B 0,C 180,E1 6510.77,E2 6510.77} C_VEL
LIN {X 0,Y 634.897,Z 977.53,A -85,B 0,C 180,E1 6515.751,E2 6515.751} C_VEL
LIN {X 0,Y 634.891,Z 977.53,A -85,B 0,C 180,E1 6520.196,E2 6520.196} C_VEL
LIN {X 0,Y 634.869,Z 977.53,A -85,B 0,C 180,E1 6525.734,E2 6525.734} C_VEL
LIN {X 0,Y 634.846,Z 977.53,A -85,B 0,C 180,E1 6531.634,E2 6531.634} C_VEL
LIN {X 0,Y 634.909,Z 977.53,A -85,B 0,C 180,E1 6536.7,E2 6536.7} C_VEL
LIN {X 0,Y 635.044,Z 977.53,A -85,B 0,C 180,E1 6541.996,E2 6541.996} C_VEL
LIN {X 0,Y 635.136,Z 977.53,A -85,B 0,C 180,E1 6547.553,E2 6547.553} C_VEL
LIN {X 0,Y 635.211,Z 977.53,A -85,B 0,C 180,E1 6553.36,E2 6553.36} C_VEL
LIN {X 0,Y 635.326,Z 977.53,A -85,B 0,C 180,E1 6558.994,E2 6558.994} C_VEL
LIN {X 0,Y 635.44,Z 977.53,A -85,B 0,C 180,E1 6564.52,E2 6564.52} C_VEL
LIN {X 0,Y 635.512,Z 977.53,A -85,B 0,C 180,E1 6568.627,E2 6568.627} C_VEL
LIN {X 0,Y 635.51,Z 977.53,A -85,B 0,C 180,E1 6572.727,E2 6572.727} C_VEL
LIN {X 0,Y 635.33,Z 977.53,A -85,B 0,C 180,E1 6576.842,E2 6576.842} C_VEL
LIN {X 0,Y 635.304,Z 977.53,A -85,B 0,C 180,E1 6582.389,E2 6582.389} C_VEL
LIN {X 0,Y 635.218,Z 977.53,A -85,B 0,C 180,E1 6588.059,E2 6588.059} C_VEL
LIN {X 0,Y 635.089,Z 977.53,A -85,B 0,C 180,E1 6592.435,E2 6592.435} C_VEL
LIN {X 0,Y 635.057,Z 977.53,A -85,B 0,C 180,E1 6598.006,E2 6598.006} C_VEL
LIN {X 0,Y 634.935,Z 977.53,A -85,B 0,C 180,E1 6603.349,E2 6603.349} C_VEL
LIN {X 0,Y 634.923,Z 977.53,A -85,B 0,C 180,E1 6608.344,E2 6608.344} C_VEL
LIN {X 0,Y 634.897,Z 977.53,A -85,B 0,C 180,E1 6613.789,E2 6613.789} C_VEL
LIN {X 0,Y 634.846,Z 977.53,A -85,B 0,C 180,E1 6619.789,E2 6619.789} C_VEL
LIN {X 0,Y 634.844,Z 977.53,A -85,B 0,C 180,E1 6625.044,E2 6625.044} C_VEL
LIN {X 0,Y 634.971,Z 977.53,A -85,B 0,C 180,E1 6629.918,E2 6629.918} C_VEL
LIN {X 0,Y 635.139,Z 977.53,A -85,B 0,C 180,E1 6632.328,E2 6632.328} C_VEL
LIN {X 0,Y 646.811,Z 1012.254,A -85,B 0,C 180,E1 6633.337,E2 6633.337} C_VEL
LIN {X 0,Y 645.742,Z 1052.007,A -85,B 0,C 180,E1 6634.315,E2 6634.315} C_VEL
LIN {X 0,Y 644.098,Z 1087.823,A -85,B 0,C 180,E1 6635.681,E2 6635.681} C_VEL
LIN {X 0,Y 642.103,Z 1122.689,A -85,B 0,C 180,E1 6637.552,E2 6637.552} C_VEL
LIN {X 0,Y 640.11,Z 1155.281,A -85,B 0,C 180,E1 6639.918,E2 6639.918} C_VEL
LIN {X 0,Y 638.403,Z 1182.778,A -85,B 0,C 180,E1 6642.555,E2 6642.555} C_VEL
LIN {X 0,Y 637.146,Z 1206.367,A -85,B 0,C 180,E1 6645.531,E2 6645.531} C_VEL
LIN {X 0,Y 636.373,Z 1224.972,A -85,B 0,C 180,E1 6648.663,E2 6648.663} C_VEL
LIN {X 0,Y 635.979,Z 1239.463,A -85,B 0,C 180,E1 6652.117,E2 6652.117} C_VEL
LIN {X 0,Y 635.772,Z 1247.786,A -85,B 0,C 180,E1 6655.206,E2 6655.206} C_VEL
LIN {X 0,Y 635.692,Z 1252.111,A -85,B 0,C 180,E1 6658.625,E2 6658.625} C_VEL
LIN {X 0,Y 635.836,Z 1252.058,A -85,B 0,C 180,E1 6661.356,E2 6661.356} C_VEL
LIN {X 0,Y 635.814,Z 1247.642,A -85,B 0,C 180,E1 6664.774,E2 6664.774} C_VEL
LIN {X 0,Y 635.987,Z 1238.089,A -85,B 0,C 180,E1 6668.208,E2 6668.208} C_VEL
LIN {X 0,Y 636.464,Z 1222.881,A -85,B 0,C 180,E1 6671.664,E2 6671.664} C_VEL
LIN {X 0,Y 637.355,Z 1202.223,A -85,B 0,C 180,E1 6674.972,E2 6674.972} C_VEL
LIN {X 0,Y 638.754,Z 1177.227,A -85,B 0,C 180,E1 6677.95,E2 6677.95} C_VEL
LIN {X 0,Y 640.558,Z 1147.786,A -85,B 0,C 180,E1 6680.589,E2 6680.589} C_VEL
LIN {X 0,Y 642.387,Z 1115.291,A -85,B 0,C 180,E1 6682.776,E2 6682.776} C_VEL
LIN {X 0,Y 644.219,Z 1078.764,A -85,B 0,C 180,E1 6684.57,E2 6684.57} C_VEL
LIN {X 0,Y 645.778,Z 1039.756,A -85,B 0,C 180,E1 6685.872,E2 6685.872} C_VEL
LIN {X 0,Y 645.867,Z 1009.194,A -85,B 0,C 180,E1 6686.545,E2 6686.545} C_VEL
LIN {X 0,Y 640.524,Z 995.199,A -85,B 0,C 180,E1 6686.945,E2 6686.945} C_VEL
LIN {X 0,Y 633.381,Z 986.354,A -85,B 0,C 180,E1 6687.328,E2 6687.328} C_VEL
LIN {X 0,Y 627.187,Z 978.29,A -85,B 0,C 180,E1 6687.692,E2 6687.692} C_VEL
LIN {X 0,Y 627.083,Z 977.662,A -85,B 0,C 180,E1 6687.72,E2 6687.72} C_VEL
LIN {X 0,Y 626.999,Z 977.53,A -85,B 0,C 180,E1 6692.25,E2 6692.25} C_VEL
LIN {X 0,Y 626.966,Z 977.53,A -85,B 0,C 180,E1 6697.154,E2 6697.154} C_VEL
LIN {X 0,Y 626.759,Z 977.53,A -85,B 0,C 180,E1 6702.585,E2 6702.585} C_VEL
LIN {X 0,Y 626.752,Z 977.53,A -85,B 0,C 180,E1 6707.404,E2 6707.404} C_VEL
LIN {X 0,Y 627.025,Z 977.53,A -85,B 0,C 180,E1 6712.864,E2 6712.864} C_VEL
LIN {X 0,Y 626.964,Z 977.53,A -85,B 0,C 180,E1 6717.887,E2 6717.887} C_VEL
LIN {X 0,Y 627.065,Z 978.049,A -85,B 0,C 180,E1 6719.719,E2 6719.719} C_VEL
LIN {X 0,Y 636.42,Z 1012.776,A -85,B 0,C 180,E1 6721.978,E2 6721.978} C_VEL
LIN {X 0,Y 639.941,Z 1021.518,A -85,B 0,C 180,E1 6722.565,E2 6722.565} C_VEL
LIN {X 0,Y 638.656,Z 1079.149,A -85,B 0,C 180,E1 6723.403,E2 6723.403} C_VEL
LIN {X 0,Y 637.221,Z 1119.513,A -85,B 0,C 180,E1 6724.538,E2 6724.538} C_VEL
LIN {X 0,Y 635.342,Z 1157.396,A -85,B 0,C 180,E1 6726.148,E2 6726.148} C_VEL
LIN {X 0,Y 633.398,Z 1192.91,A -85,B 0,C 180,E1 6728.242,E2 6728.242} C_VEL
LIN {X 0,Y 631.461,Z 1226.838,A -85,B 0,C 180,E1 6730.935,E2 6730.935} C_VEL
LIN {X 0,Y 629.877,Z 1254.77,A -85,B 0,C 180,E1 6733.904,E2 6733.904} C_VEL
LIN {X 0,Y 628.897,Z 1275.182,A -85,B 0,C 180,E1 6736.775,E2 6736.775} C_VEL
LIN {X 0,Y 628.29,Z 1291.393,A -85,B 0,C 180,E1 6739.937,E2 6739.937} C_VEL
LIN {X 0,Y 627.958,Z 1302.589,A -85,B 0,C 180,E1 6743.077,E2 6743.077} C_VEL
LIN {X 0,Y 627.842,Z 1308.95,A -85,B 0,C 180,E1 6745.854,E2 6745.854} C_VEL
LIN {X 0,Y 627.873,Z 1312.102,A -85,B 0,C 180,E1 6748.624,E2 6748.624} C_VEL
LIN {X 0,Y 627.876,Z 1312.1,A -85,B 0,C 180,E1 6751.389,E2 6751.389} C_VEL
LIN {X 0,Y 627.944,Z 1307.632,A -85,B 0,C 180,E1 6754.851,E2 6754.851} C_VEL
LIN {X 0,Y 628.134,Z 1297.201,A -85,B 0,C 180,E1 6758.597,E2 6758.597} C_VEL
LIN {X 0,Y 628.669,Z 1281.059,A -85,B 0,C 180,E1 6762.182,E2 6762.182} C_VEL
LIN {X 0,Y 629.523,Z 1261.954,A -85,B 0,C 180,E1 6765.181,E2 6765.181} C_VEL
LIN {X 0,Y 630.765,Z 1237.208,A -85,B 0,C 180,E1 6768.023,E2 6768.023} C_VEL
LIN {X 0,Y 632.514,Z 1205.629,A -85,B 0,C 180,E1 6770.756,E2 6770.756} C_VEL
LIN {X 0,Y 634.471,Z 1169.707,A -85,B 0,C 180,E1 6773.1,E2 6773.1} C_VEL
LIN {X 0,Y 636.452,Z 1132.503,A -85,B 0,C 180,E1 6774.898,E2 6774.898} C_VEL
LIN {X 0,Y 638.026,Z 1094.242,A -85,B 0,C 180,E1 6776.165,E2 6776.165} C_VEL
LIN {X 0,Y 639.042,Z 1053.962,A -85,B 0,C 180,E1 6776.948,E2 6776.948} C_VEL
LIN {X 0,Y 638.987,Z 1018.019,A -85,B 0,C 180,E1 6777.405,E2 6777.405} C_VEL
LIN {X 0,Y 630.99,Z 997.658,A -85,B 0,C 180,E1 6778.67,E2 6778.67} C_VEL
LIN {X 0,Y 627.105,Z 977.53,A -85,B 0,C 180,E1 6779.903,E2 6779.903} C_VEL
LIN {X 0,Y 627.014,Z 977.53,A -85,B 0,C 180,E1 6785.458,E2 6785.458} C_VEL
LIN {X 0,Y 626.93,Z 977.53,A -85,B 0,C 180,E1 6790.745,E2 6790.745} C_VEL
LIN {X 0,Y 626.996,Z 977.53,A -85,B 0,C 180,E1 6795.526,E2 6795.526} C_VEL
LIN {X 0,Y 626.877,Z 977.53,A -85,B 0,C 180,E1 6801.081,E2 6801.081} C_VEL
LIN {X 0,Y 626.932,Z 977.53,A -85,B 0,C 180,E1 6806.244,E2 6806.244} C_VEL
LIN {X 0,Y 627.095,Z 977.53,A -85,B 0,C 180,E1 6811.116,E2 6811.116} C_VEL
LIN {X 0,Y 627.175,Z 977.53,A -85,B 0,C 180,E1 6816.664,E2 6816.664} C_VEL
LIN {X 0,Y 627.277,Z 977.53,A -85,B 0,C 180,E1 6821.71,E2 6821.71} C_VEL
LIN {X 0,Y 627.275,Z 977.53,A -85,B 0,C 180,E1 6827.455,E2 6827.455} C_VEL
LIN {X 0,Y 627.561,Z 977.53,A -85,B 0,C 180,E1 6833.077,E2 6833.077} C_VEL
LIN {X 0,Y 627.596,Z 978.286,A -85,B 0,C 180,E1 6834.425,E2 6834.425} C_VEL
LIN {X 0,Y 633.281,Z 1000.746,A -85,B 0,C 180,E1 6835.006,E2 6835.006} C_VEL
LIN {X 0,Y 632.486,Z 1057.039,A -85,B 0,C 180,E1 6835.975,E2 6835.975} C_VEL
LIN {X 0,Y 631.765,Z 1085.127,A -85,B 0,C 180,E1 6837.003,E2 6837.003} C_VEL
LIN {X 0,Y 630.907,Z 1110.84,A -85,B 0,C 180,E1 6838.548,E2 6838.548} C_VEL
LIN {X 0,Y 629.963,Z 1132.878,A -85,B 0,C 180,E1 6840.527,E2 6840.527} C_VEL
LIN {X 0,Y 629.263,Z 1149.7,A -85,B 0,C 180,E1 6842.77,E2 6842.77} C_VEL
LIN {X 0,Y 628.746,Z 1161.41,A -85,B 0,C 180,E1 6845.194,E2 6845.194} C_VEL
LIN {X 0,Y 628.44,Z 1167.904,A -85,B 0,C 180,E1 6847.63,E2 6847.63} C_VEL
LIN {X 0,Y 628.33,Z 1169.743,A -85,B 0,C 180,E1 6849.727,E2 6849.727} C_VEL
LIN {X 0,Y 628.444,Z 1166.977,A -85,B 0,C 180,E1 6852.542,E2 6852.542} C_VEL
LIN {X 0,Y 628.705,Z 1159.284,A -85,B 0,C 180,E1 6855.024,E2 6855.024} C_VEL
LIN {X 0,Y 629.105,Z 1145.476,A -85,B 0,C 180,E1 6857.56,E2 6857.56} C_VEL
LIN {X 0,Y 629.848,Z 1126.292,A -85,B 0,C 180,E1 6859.837,E2 6859.837} C_VEL
LIN {X 0,Y 630.653,Z 1102.676,A -85,B 0,C 180,E1 6861.714,E2 6861.714} C_VEL
LIN {X 0,Y 631.584,Z 1075.211,A -85,B 0,C 180,E1 6863.14,E2 6863.14} C_VEL
LIN {X 0,Y 632.069,Z 1046.56,A -85,B 0,C 180,E1 6864.011,E2 6864.011} C_VEL
LIN {X 0,Y 631.644,Z 994.273,A -85,B 0,C 180,E1 6864.784,E2 6864.784} C_VEL
LIN {X 0,Y 627.333,Z 977.53,A -85,B 0,C 180,E1 6865.199,E2 6865.199} C_VEL
LIN {X 0,Y 627.06,Z 977.53,A -85,B 0,C 180,E1 6870.502,E2 6870.502} C_VEL
LIN {X 0,Y 626.982,Z 977.53,A -85,B 0,C 180,E1 6875.459,E2 6875.459} C_VEL
LIN {X 0,Y 626.951,Z 977.53,A -85,B 0,C 180,E1 6880.742,E2 6880.742} C_VEL
LIN {X 0,Y 626.974,Z 977.53,A -85,B 0,C 180,E1 6885.494,E2 6885.494} C_VEL
LIN {X 0,Y 626.87,Z 977.53,A -85,B 0,C 180,E1 6891.055,E2 6891.055} C_VEL
LIN {X 0,Y 626.954,Z 977.53,A -85,B 0,C 180,E1 6896.221,E2 6896.221} C_VEL
LIN {X 0,Y 627.067,Z 977.53,A -85,B 0,C 180,E1 6901.092,E2 6901.092} C_VEL
LIN {X 0,Y 627.19,Z 977.53,A -85,B 0,C 180,E1 6906.654,E2 6906.654} C_VEL
LIN {X 0,Y 627.253,Z 977.53,A -85,B 0,C 180,E1 6911.69,E2 6911.69} C_VEL
LIN {X 0,Y 627.264,Z 977.53,A -85,B 0,C 180,E1 6916.014,E2 6916.014} C_VEL
LIN {X 0,Y 627.486,Z 977.53,A -85,B 0,C 180,E1 6921.663,E2 6921.663} C_VEL
LIN {X 0,Y 627.666,Z 977.53,A -85,B 0,C 180,E1 6927.226,E2 6927.226} C_VEL
LIN {X 0,Y 627.607,Z 977.53,A -85,B 0,C 180,E1 6932.761,E2 6932.761} C_VEL
LIN {X 0,Y 627.447,Z 977.53,A -85,B 0,C 180,E1 6938.031,E2 6938.031} C_VEL
LIN {X 0,Y 627.381,Z 977.53,A -85,B 0,C 180,E1 6942.548,E2 6942.548} C_VEL
LIN {X 0,Y 627.289,Z 977.53,A -85,B 0,C 180,E1 6948.295,E2 6948.295} C_VEL
LIN {X 0,Y 627.123,Z 977.53,A -85,B 0,C 180,E1 6953.332,E2 6953.332} C_VEL
LIN {X 0,Y 627.09,Z 977.53,A -85,B 0,C 180,E1 6958.892,E2 6958.892} C_VEL
LIN {X 0,Y 626.992,Z 977.53,A -85,B 0,C 180,E1 6964.739,E2 6964.739} C_VEL
LIN {X 0,Y 626.941,Z 977.53,A -85,B 0,C 180,E1 6969.331,E2 6969.331} C_VEL
LIN {X 0,Y 626.978,Z 977.53,A -85,B 0,C 180,E1 6974.487,E2 6974.487} C_VEL
LIN {X 0,Y 626.897,Z 977.53,A -85,B 0,C 180,E1 6979.254,E2 6979.254} C_VEL
LIN {X 0,Y 626.936,Z 977.53,A -85,B 0,C 180,E1 6984.538,E2 6984.538} C_VEL
LIN {X 0,Y 627.062,Z 977.53,A -85,B 0,C 180,E1 6990.436,E2 6990.436} C_VEL
LIN {X 0,Y 627.276,Z 978.271,A -85,B 0,C 180,E1 6992.027,E2 6992.027} C_VEL
LIN {X 0,Y 639.618,Z 1012.612,A -85,B 0,C 180,E1 6993.052,E2 6993.052} C_VEL
LIN {X 0,Y 638.423,Z 1053.217,A -85,B 0,C 180,E1 6994.069,E2 6994.069} C_VEL
LIN {X 0,Y 636.678,Z 1089.196,A -85,B 0,C 180,E1 6995.473,E2 6995.473} C_VEL
LIN {X 0,Y 634.537,Z 1124.639,A -85,B 0,C 180,E1 6997.419,E2 6997.419} C_VEL
LIN {X 0,Y 632.466,Z 1156.291,A -85,B 0,C 180,E1 6999.763,E2 6999.763} C_VEL
LIN {X 0,Y 630.629,Z 1184.377,A -85,B 0,C 180,E1 7002.513,E2 7002.513} C_VEL
LIN {X 0,Y 629.327,Z 1207.599,A -85,B 0,C 180,E1 7005.526,E2 7005.526} C_VEL
LIN {X 0,Y 628.419,Z 1226.698,A -85,B 0,C 180,E1 7008.869,E2 7008.869} C_VEL
LIN {X 0,Y 628.075,Z 1240.604,A -85,B 0,C 180,E1 7012.366,E2 7012.366} C_VEL
LIN {X 0,Y 627.816,Z 1248.99,A -85,B 0,C 180,E1 7015.838,E2 7015.838} C_VEL
LIN {X 0,Y 627.791,Z 1252.111,A -85,B 0,C 180,E1 7018.607,E2 7018.607} C_VEL
LIN {X 0,Y 627.934,Z 1252.058,A -85,B 0,C 180,E1 7021.373,E2 7021.373} C_VEL
LIN {X 0,Y 627.937,Z 1247.643,A -85,B 0,C 180,E1 7024.834,E2 7024.834} C_VEL
LIN {X 0,Y 628.141,Z 1237.273,A -85,B 0,C 180,E1 7028.534,E2 7028.534} C_VEL
LIN {X 0,Y 628.674,Z 1220.953,A -85,B 0,C 180,E1 7032.163,E2 7032.163} C_VEL
LIN {X 0,Y 629.684,Z 1200.985,A -85,B 0,C 180,E1 7035.337,E2 7035.337} C_VEL
LIN {X 0,Y 631.169,Z 1175.845,A -85,B 0,C 180,E1 7038.313,E2 7038.313} C_VEL
LIN {X 0,Y 633.076,Z 1146.452,A -85,B 0,C 180,E1 7040.928,E2 7040.928} C_VEL
LIN {X 0,Y 635.022,Z 1113.749,A -85,B 0,C 180,E1 7043.113,E2 7043.113} C_VEL
LIN {X 0,Y 636.872,Z 1077.653,A -85,B 0,C 180,E1 7044.873,E2 7044.873} C_VEL
LIN {X 0,Y 638.522,Z 1036.849,A -85,B 0,C 180,E1 7046.215,E2 7046.215} C_VEL
LIN {X 0,Y 638.536,Z 1011.239,A -85,B 0,C 180,E1 7046.779,E2 7046.779} C_VEL
LIN {X 0,Y 627.083,Z 977.662,A -85,B 0,C 180,E1 7047.72,E2 7047.72} C_VEL
LIN {X 0,Y 625.614,Z 973.822,A -85,B 0,C 180,E1 7048.22,E2 7048.22} C_VEL
LIN {X 0,Y 622.69,Z 973.749,A -85,B 0,C 180,E1 7049.066,E2 7049.066} C_VEL
LIN {X 0,Y 619.117,Z 977.416,A -85,B 0,C 180,E1 7050.624,E2 7050.624} C_VEL
LIN {X 0,Y 619.06,Z 977.53,A -85,B 0,C 180,E1 7050.856,E2 7050.856} C_VEL
LIN {X 0,Y 619.014,Z 977.53,A -85,B 0,C 180,E1 7056.13,E2 7056.13} C_VEL
LIN {X 0,Y 618.882,Z 977.53,A -85,B 0,C 180,E1 7061.362,E2 7061.362} C_VEL
LIN {X 0,Y 618.842,Z 977.53,A -85,B 0,C 180,E1 7067.248,E2 7067.248} C_VEL
LIN {X 0,Y 619.022,Z 977.53,A -85,B 0,C 180,E1 7072.277,E2 7072.277} C_VEL
LIN {X 0,Y 619.051,Z 977.53,A -85,B 0,C 180,E1 7077.426,E2 7077.426} C_VEL
LIN {X 0,Y 619.136,Z 978.146,A -85,B 0,C 180,E1 7079.399,E2 7079.399} C_VEL
LIN {X 0,Y 629.16,Z 1015.664,A -85,B 0,C 180,E1 7081.874,E2 7081.874} C_VEL
LIN {X 0,Y 632.39,Z 1022.242,A -85,B 0,C 180,E1 7082.306,E2 7082.306} C_VEL
LIN {X 0,Y 631.359,Z 1077.985,A -85,B 0,C 180,E1 7083.119,E2 7083.119} C_VEL
LIN {X 0,Y 629.812,Z 1118.092,A -85,B 0,C 180,E1 7084.25,E2 7084.25} C_VEL
LIN {X 0,Y 627.799,Z 1156.705,A -85,B 0,C 180,E1 7085.906,E2 7085.906} C_VEL
LIN {X 0,Y 625.689,Z 1192.631,A -85,B 0,C 180,E1 7088.053,E2 7088.053} C_VEL
LIN {X 0,Y 623.776,Z 1225.135,A -85,B 0,C 180,E1 7090.657,E2 7090.657} C_VEL
LIN {X 0,Y 622.2,Z 1252.035,A -85,B 0,C 180,E1 7093.501,E2 7093.501} C_VEL
LIN {X 0,Y 620.995,Z 1275.528,A -85,B 0,C 180,E1 7096.783,E2 7096.783} C_VEL
LIN {X 0,Y 620.429,Z 1291.356,A -85,B 0,C 180,E1 7099.808,E2 7099.808} C_VEL
LIN {X 0,Y 620.08,Z 1302.588,A -85,B 0,C 180,E1 7102.988,E2 7102.988} C_VEL
LIN {X 0,Y 619.948,Z 1308.945,A -85,B 0,C 180,E1 7105.802,E2 7105.802} C_VEL
LIN {X 0,Y 619.998,Z 1312.098,A -85,B 0,C 180,E1 7108.606,E2 7108.606} C_VEL
LIN {X 0,Y 620.001,Z 1312.097,A -85,B 0,C 180,E1 7111.407,E2 7111.407} C_VEL
LIN {X 0,Y 620.06,Z 1307.628,A -85,B 0,C 180,E1 7114.913,E2 7114.913} C_VEL
LIN {X 0,Y 620.234,Z 1297.197,A -85,B 0,C 180,E1 7118.707,E2 7118.707} C_VEL
LIN {X 0,Y 620.761,Z 1282.766,A -85,B 0,C 180,E1 7121.944,E2 7121.944} C_VEL
LIN {X 0,Y 621.706,Z 1260.591,A -85,B 0,C 180,E1 7125.377,E2 7125.377} C_VEL
LIN {X 0,Y 623.033,Z 1235.588,A -85,B 0,C 180,E1 7128.255,E2 7128.255} C_VEL
LIN {X 0,Y 625.042,Z 1201.269,A -85,B 0,C 180,E1 7131.237,E2 7131.237} C_VEL
LIN {X 0,Y 627.157,Z 1166.622,A -85,B 0,C 180,E1 7133.511,E2 7133.511} C_VEL
LIN {X 0,Y 629.194,Z 1129.927,A -85,B 0,C 180,E1 7135.265,E2 7135.265} C_VEL
LIN {X 0,Y 630.901,Z 1089.141,A -85,B 0,C 180,E1 7136.579,E2 7136.579} C_VEL
LIN {X 0,Y 631.852,Z 1048.338,A -85,B 0,C 180,E1 7137.317,E2 7137.317} C_VEL
LIN {X 0,Y 631.452,Z 1020.238,A -85,B 0,C 180,E1 7137.694,E2 7137.694} C_VEL
LIN {X 0,Y 626.5,Z 1009.667,A -85,B 0,C 180,E1 7138.179,E2 7138.179} C_VEL
LIN {X 0,Y 619.167,Z 977.53,A -85,B 0,C 180,E1 7140.233,E2 7140.233} C_VEL
LIN {X 0,Y 619.047,Z 977.53,A -85,B 0,C 180,E1 7145.985,E2 7145.985} C_VEL
LIN {X 0,Y 619.023,Z 977.53,A -85,B 0,C 180,E1 7151.378,E2 7151.378} C_VEL
LIN {X 0,Y 619.008,Z 977.53,A -85,B 0,C 180,E1 7156.752,E2 7156.752} C_VEL
LIN {X 0,Y 618.951,Z 977.53,A -85,B 0,C 180,E1 7162.282,E2 7162.282} C_VEL
LIN {X 0,Y 619.034,Z 977.53,A -85,B 0,C 180,E1 7167.434,E2 7167.434} C_VEL
LIN {X 0,Y 619.215,Z 977.53,A -85,B 0,C 180,E1 7172.308,E2 7172.308} C_VEL
LIN {X 0,Y 619.294,Z 977.53,A -85,B 0,C 180,E1 7176.967,E2 7176.967} C_VEL
LIN {X 0,Y 619.337,Z 977.53,A -85,B 0,C 180,E1 7182.608,E2 7182.608} C_VEL
LIN {X 0,Y 619.377,Z 977.53,A -85,B 0,C 180,E1 7188.149,E2 7188.149} C_VEL
LIN {X 0,Y 619.654,Z 977.53,A -85,B 0,C 180,E1 7193.693,E2 7193.693} C_VEL
LIN {X 0,Y 619.625,Z 977.53,A -85,B 0,C 180,E1 7194.089,E2 7194.089} C_VEL
LIN {X 0,Y 625.875,Z 1002.191,A -85,B 0,C 180,E1 7194.77,E2 7194.77} C_VEL
LIN {X 0,Y 625.014,Z 1057.428,A -85,B 0,C 180,E1 7195.751,E2 7195.751} C_VEL
LIN {X 0,Y 624.231,Z 1085.708,A -85,B 0,C 180,E1 7196.792,E2 7196.792} C_VEL
LIN {X 0,Y 623.321,Z 1111.522,A -85,B 0,C 180,E1 7198.356,E2 7198.356} C_VEL
LIN {X 0,Y 622.281,Z 1133.62,A -85,B 0,C 180,E1 7200.359,E2 7200.359} C_VEL
LIN {X 0,Y 621.526,Z 1150.391,A -85,B 0,C 180,E1 7202.612,E2 7202.612} C_VEL
LIN {X 0,Y 620.928,Z 1162.867,A -85,B 0,C 180,E1 7205.26,E2 7205.26} C_VEL
LIN {X 0,Y 620.592,Z 1169.076,A -85,B 0,C 180,E1 7207.727,E2 7207.727} C_VEL
LIN {X 0,Y 620.498,Z 1170.706,A -85,B 0,C 180,E1 7209.851,E2 7209.851} C_VEL
LIN {X 0,Y 620.615,Z 1167.591,A -85,B 0,C 180,E1 7212.702,E2 7212.702} C_VEL
LIN {X 0,Y 620.899,Z 1159.718,A -85,B 0,C 180,E1 7215.189,E2 7215.189} C_VEL
LIN {X 0,Y 621.353,Z 1145.62,A -85,B 0,C 180,E1 7217.759,E2 7217.759} C_VEL
LIN {X 0,Y 622.101,Z 1127.282,A -85,B 0,C 180,E1 7219.946,E2 7219.946} C_VEL
LIN {X 0,Y 622.941,Z 1104.042,A -85,B 0,C 180,E1 7221.827,E2 7221.827} C_VEL
LIN {X 0,Y 623.941,Z 1077.389,A -85,B 0,C 180,E1 7223.251,E2 7223.251} C_VEL
LIN {X 0,Y 624.492,Z 1048.172,A -85,B 0,C 180,E1 7224.178,E2 7224.178} C_VEL
LIN {X 0,Y 624.177,Z 995.839,A -85,B 0,C 180,E1 7224.974,E2 7224.974} C_VEL
LIN {X 0,Y 619.387,Z 977.53,A -85,B 0,C 180,E1 7225.425,E2 7225.425} C_VEL
LIN {X 0,Y 619.102,Z 977.53,A -85,B 0,C 180,E1 7231.047,E2 7231.047} C_VEL
LIN {X 0,Y 619.026,Z 977.53,A -85,B 0,C 180,E1 7236.109,E2 7236.109} C_VEL
LIN {X 0,Y 619.047,Z 977.53,A -85,B 0,C 180,E1 7241.375,E2 7241.375} C_VEL
LIN {X 0,Y 619.017,Z 977.53,A -85,B 0,C 180,E1 7246.724,E2 7246.724} C_VEL
LIN {X 0,Y 618.95,Z 977.53,A -85,B 0,C 180,E1 7252.255,E2 7252.255} C_VEL
LIN {X 0,Y 619.069,Z 977.53,A -85,B 0,C 180,E1 7257.412,E2 7257.412} C_VEL
LIN {X 0,Y 619.197,Z 977.53,A -85,B 0,C 180,E1 7262.285,E2 7262.285} C_VEL
LIN {X 0,Y 619.287,Z 977.53,A -85,B 0,C 180,E1 7266.946,E2 7266.946} C_VEL
LIN {X 0,Y 619.364,Z 977.53,A -85,B 0,C 180,E1 7272.59,E2 7272.59} C_VEL
LIN {X 0,Y 619.435,Z 977.53,A -85,B 0,C 180,E1 7278.109,E2 7278.109} C_VEL
LIN {X 0,Y 619.664,Z 977.53,A -85,B 0,C 180,E1 7282.971,E2 7282.971} C_VEL
LIN {X 0,Y 619.711,Z 977.53,A -85,B 0,C 180,E1 7288.592,E2 7288.592} C_VEL
LIN {X 0,Y 619.735,Z 977.53,A -85,B 0,C 180,E1 7292.796,E2 7292.796} C_VEL
LIN {X 0,Y 619.534,Z 977.53,A -85,B 0,C 180,E1 7297.018,E2 7297.018} C_VEL
LIN {X 0,Y 619.463,Z 977.53,A -85,B 0,C 180,E1 7302.711,E2 7302.711} C_VEL
LIN {X 0,Y 619.365,Z 977.53,A -85,B 0,C 180,E1 7307.41,E2 7307.41} C_VEL
LIN {X 0,Y 619.228,Z 977.53,A -85,B 0,C 180,E1 7313.042,E2 7313.042} C_VEL
LIN {X 0,Y 619.157,Z 977.53,A -85,B 0,C 180,E1 7318.225,E2 7318.225} C_VEL
LIN {X 0,Y 619.09,Z 977.53,A -85,B 0,C 180,E1 7323.67,E2 7323.67} C_VEL
LIN {X 0,Y 619.02,Z 977.53,A -85,B 0,C 180,E1 7329.518,E2 7329.518} C_VEL
LIN {X 0,Y 619.048,Z 977.53,A -85,B 0,C 180,E1 7335.213,E2 7335.213} C_VEL
LIN {X 0,Y 618.972,Z 977.53,A -85,B 0,C 180,E1 7340.462,E2 7340.462} C_VEL
LIN {X 0,Y 619.03,Z 977.53,A -85,B 0,C 180,E1 7346.319,E2 7346.319} C_VEL
LIN {X 0,Y 619.287,Z 977.53,A -85,B 0,C 180,E1 7351.651,E2 7351.651} C_VEL
LIN {X 0,Y 632.366,Z 1015.698,A -85,B 0,C 180,E1 7352.814,E2 7352.814} C_VEL
LIN {X 0,Y 631.026,Z 1055.667,A -85,B 0,C 180,E1 7353.858,E2 7353.858} C_VEL
LIN {X 0,Y 629.127,Z 1092.537,A -85,B 0,C 180,E1 7355.353,E2 7355.353} C_VEL
LIN {X 0,Y 626.938,Z 1127.383,A -85,B 0,C 180,E1 7357.336,E2 7357.336} C_VEL
LIN {X 0,Y 624.704,Z 1159.677,A -85,B 0,C 180,E1 7359.812,E2 7359.812} C_VEL
LIN {X 0,Y 622.688,Z 1189.074,A -85,B 0,C 180,E1 7362.831,E2 7362.831} C_VEL
LIN {X 0,Y 621.311,Z 1212.302,A -85,B 0,C 180,E1 7366.056,E2 7366.056} C_VEL
LIN {X 0,Y 620.468,Z 1230.024,A -85,B 0,C 180,E1 7369.437,E2 7369.437} C_VEL
LIN {X 0,Y 620.079,Z 1242.701,A -85,B 0,C 180,E1 7372.973,E2 7372.973} C_VEL
LIN {X 0,Y 619.927,Z 1248.989,A -85,B 0,C 180,E1 7375.785,E2 7375.785} C_VEL
LIN {X 0,Y 619.904,Z 1252.111,A -85,B 0,C 180,E1 7378.59,E2 7378.59} C_VEL
LIN {X 0,Y 620.043,Z 1252.058,A -85,B 0,C 180,E1 7381.39,E2 7381.39} C_VEL
LIN {X 0,Y 620.066,Z 1247.644,A -85,B 0,C 180,E1 7384.896,E2 7384.896} C_VEL
LIN {X 0,Y 620.251,Z 1237.274,A -85,B 0,C 180,E1 7388.644,E2 7388.644} C_VEL
LIN {X 0,Y 620.837,Z 1221.516,A -85,B 0,C 180,E1 7392.247,E2 7392.247} C_VEL
LIN {X 0,Y 621.975,Z 1201.111,A -85,B 0,C 180,E1 7395.532,E2 7395.532} C_VEL
LIN {X 0,Y 623.51,Z 1176.206,A -85,B 0,C 180,E1 7398.503,E2 7398.503} C_VEL
LIN {X 0,Y 625.434,Z 1147.703,A -85,B 0,C 180,E1 7401.073,E2 7401.073} C_VEL
LIN {X 0,Y 627.511,Z 1114.327,A -85,B 0,C 180,E1 7403.333,E2 7403.333} C_VEL
LIN {X 0,Y 629.491,Z 1077.769,A -85,B 0,C 180,E1 7405.131,E2 7405.131} C_VEL
LIN {X 0,Y 631.182,Z 1037.196,A -85,B 0,C 180,E1 7406.479,E2 7406.479} C_VEL
LIN {X 0,Y 631.319,Z 1013.579,A -85,B 0,C 180,E1 7407.008,E2 7407.008} C_VEL
LIN {X 0,Y 619.189,Z 977.53,A -85,B 0,C 180,E1 7408.09,E2 7408.09} C_VEL
LIN {X 0,Y 619.06,Z 977.53,A -85,B 0,C 180,E1 7410.856,E2 7410.856} C_VEL
LIN {X 0,Y 616.577,Z 977.53,A -85,B 0,C 180,E1 7412.052,E2 7412.052} C_VEL
LIN {X 0,Y 611.15,Z 977.53,A -85,B 0,C 180,E1 7413.841,E2 7413.841} C_VEL
LIN {X 0,Y 611.055,Z 977.53,A -85,B 0,C 180,E1 7414.047,E2 7414.047} C_VEL
LIN {X 0,Y 611.036,Z 977.53,A -85,B 0,C 180,E1 7419.769,E2 7419.769} C_VEL
LIN {X 0,Y 610.909,Z 977.53,A -85,B 0,C 180,E1 7426.022,E2 7426.022} C_VEL
LIN {X 0,Y 611.081,Z 977.53,A -85,B 0,C 180,E1 7431.699,E2 7431.699} C_VEL
LIN {X 0,Y 611.174,Z 977.53,A -85,B 0,C 180,E1 7437.424,E2 7437.424} C_VEL
LIN {X 0,Y 611.19,Z 978.022,A -85,B 0,C 180,E1 7439.062,E2 7439.062} C_VEL
LIN {X 0,Y 622.016,Z 1018.92,A -85,B 0,C 180,E1 7441.791,E2 7441.791} C_VEL
LIN {X 0,Y 624.982,Z 1024.717,A -85,B 0,C 180,E1 7442.047,E2 7442.047} C_VEL
LIN {X 0,Y 624.067,Z 1076.825,A -85,B 0,C 180,E1 7442.828,E2 7442.828} C_VEL
LIN {X 0,Y 622.336,Z 1118.281,A -85,B 0,C 180,E1 7444.014,E2 7444.014} C_VEL
LIN {X 0,Y 620.208,Z 1156.611,A -85,B 0,C 180,E1 7445.688,E2 7445.688} C_VEL
LIN {X 0,Y 617.996,Z 1192.378,A -85,B 0,C 180,E1 7447.86,E2 7447.86} C_VEL
LIN {X 0,Y 615.92,Z 1226.022,A -85,B 0,C 180,E1 7450.609,E2 7450.609} C_VEL
LIN {X 0,Y 614.187,Z 1254.443,A -85,B 0,C 180,E1 7453.728,E2 7453.728} C_VEL
LIN {X 0,Y 613.058,Z 1276.617,A -85,B 0,C 180,E1 7456.972,E2 7456.972} C_VEL
LIN {X 0,Y 612.407,Z 1293.458,A -85,B 0,C 180,E1 7460.392,E2 7460.392} C_VEL
LIN {X 0,Y 612.183,Z 1304.281,A -85,B 0,C 180,E1 7463.612,E2 7463.612} C_VEL
LIN {X 0,Y 612.04,Z 1310.9,A -85,B 0,C 180,E1 7467.168,E2 7467.168} C_VEL
LIN {X 0,Y 612.031,Z 1312.5,A -85,B 0,C 180,E1 7470.007,E2 7470.007} C_VEL
LIN {X 0,Y 612.016,Z 1309.948,A -85,B 0,C 180,E1 7473.555,E2 7473.555} C_VEL
LIN {X 0,Y 612.206,Z 1302.218,A -85,B 0,C 180,E1 7477.115,E2 7477.115} C_VEL
LIN {X 0,Y 612.645,Z 1288.637,A -85,B 0,C 180,E1 7480.697,E2 7480.697} C_VEL
LIN {X 0,Y 613.491,Z 1268.276,A -85,B 0,C 180,E1 7484.306,E2 7484.306} C_VEL
LIN {X 0,Y 614.732,Z 1244.266,A -85,B 0,C 180,E1 7487.397,E2 7487.397} C_VEL
LIN {X 0,Y 616.683,Z 1212.771,A -85,B 0,C 180,E1 7490.511,E2 7490.511} C_VEL
LIN {X 0,Y 618.847,Z 1179.45,A -85,B 0,C 180,E1 7492.976,E2 7492.976} C_VEL
LIN {X 0,Y 621.066,Z 1142.909,A -85,B 0,C 180,E1 7494.971,E2 7494.971} C_VEL
LIN {X 0,Y 623.143,Z 1102.521,A -85,B 0,C 180,E1 7496.498,E2 7496.498} C_VEL
LIN {X 0,Y 624.463,Z 1062.752,A -85,B 0,C 180,E1 7497.412,E2 7497.412} C_VEL
LIN {X 0,Y 624.396,Z 1023.075,A -85,B 0,C 180,E1 7497.96,E2 7497.96} C_VEL
LIN {X 0,Y 617.654,Z 1008.278,A -85,B 0,C 180,E1 7498.536,E2 7498.536} C_VEL
LIN {X 0,Y 611.259,Z 977.53,A -85,B 0,C 180,E1 7500.535,E2 7500.535} C_VEL
LIN {X 0,Y 611.101,Z 977.53,A -85,B 0,C 180,E1 7505.117,E2 7505.117} C_VEL
LIN {X 0,Y 611.105,Z 977.53,A -85,B 0,C 180,E1 7510.15,E2 7510.15} C_VEL
LIN {X 0,Y 611.101,Z 977.53,A -85,B 0,C 180,E1 7516.051,E2 7516.051} C_VEL
LIN {X 0,Y 611.032,Z 977.53,A -85,B 0,C 180,E1 7521.705,E2 7521.705} C_VEL
LIN {X 0,Y 611.139,Z 977.53,A -85,B 0,C 180,E1 7527.47,E2 7527.47} C_VEL
LIN {X 0,Y 611.306,Z 977.53,A -85,B 0,C 180,E1 7533.184,E2 7533.184} C_VEL
LIN {X 0,Y 611.388,Z 977.53,A -85,B 0,C 180,E1 7538.189,E2 7538.189} C_VEL
LIN {X 0,Y 611.457,Z 977.53,A -85,B 0,C 180,E1 7542.713,E2 7542.713} C_VEL
LIN {X 0,Y 611.552,Z 977.53,A -85,B 0,C 180,E1 7548.579,E2 7548.579} C_VEL
LIN {X 0,Y 611.765,Z 978.051,A -85,B 0,C 180,E1 7553.79,E2 7553.79} C_VEL
LIN {X 0,Y 618.55,Z 1002.203,A -85,B 0,C 180,E1 7554.502,E2 7554.502} C_VEL
LIN {X 0,Y 617.508,Z 1059.623,A -85,B 0,C 180,E1 7555.565,E2 7555.565} C_VEL
LIN {X 0,Y 616.663,Z 1088.13,A -85,B 0,C 180,E1 7556.665,E2 7556.665} C_VEL
LIN {X 0,Y 615.606,Z 1114.522,A -85,B 0,C 180,E1 7558.335,E2 7558.335} C_VEL
LIN {X 0,Y 614.555,Z 1135.853,A -85,B 0,C 180,E1 7560.352,E2 7560.352} C_VEL
LIN {X 0,Y 613.756,Z 1152.215,A -85,B 0,C 180,E1 7562.645,E2 7562.645} C_VEL
LIN {X 0,Y 613.099,Z 1164.351,A -85,B 0,C 180,E1 7565.327,E2 7565.327} C_VEL
LIN {X 0,Y 612.836,Z 1169.041,A -85,B 0,C 180,E1 7567.111,E2 7567.111} C_VEL
LIN {X 0,Y 612.67,Z 1171.658,A -85,B 0,C 180,E1 7569.979,E2 7569.979} C_VEL
LIN {X 0,Y 612.8,Z 1168.202,A -85,B 0,C 180,E1 7572.867,E2 7572.867} C_VEL
LIN {X 0,Y 613.08,Z 1159.904,A -85,B 0,C 180,E1 7575.416,E2 7575.416} C_VEL
LIN {X 0,Y 613.597,Z 1146.194,A -85,B 0,C 180,E1 7577.899,E2 7577.899} C_VEL
LIN {X 0,Y 614.449,Z 1126.746,A -85,B 0,C 180,E1 7580.205,E2 7580.205} C_VEL
LIN {X 0,Y 615.297,Z 1103.572,A -85,B 0,C 180,E1 7582.065,E2 7582.065} C_VEL
LIN {X 0,Y 616.369,Z 1076.387,A -85,B 0,C 180,E1 7583.502,E2 7583.502} C_VEL
LIN {X 0,Y 616.87,Z 1046.701,A -85,B 0,C 180,E1 7584.415,E2 7584.415} C_VEL
LIN {X 0,Y 616.755,Z 997.76,A -85,B 0,C 180,E1 7585.164,E2 7585.164} C_VEL
LIN {X 0,Y 611.485,Z 977.53,A -85,B 0,C 180,E1 7585.686,E2 7585.686} C_VEL
LIN {X 0,Y 611.174,Z 977.53,A -85,B 0,C 180,E1 7591.383,E2 7591.383} C_VEL
LIN {X 0,Y 611.079,Z 977.53,A -85,B 0,C 180,E1 7596.529,E2 7596.529} C_VEL
LIN {X 0,Y 611.116,Z 977.53,A -85,B 0,C 180,E1 7602.033,E2 7602.033} C_VEL
LIN {X 0,Y 611.05,Z 977.53,A -85,B 0,C 180,E1 7607.96,E2 7607.96} C_VEL
LIN {X 0,Y 611.011,Z 977.53,A -85,B 0,C 180,E1 7613.466,E2 7613.466} C_VEL
LIN {X 0,Y 611.164,Z 977.53,A -85,B 0,C 180,E1 7618.616,E2 7618.616} C_VEL
LIN {X 0,Y 611.301,Z 977.53,A -85,B 0,C 180,E1 7623.494,E2 7623.494} C_VEL
LIN {X 0,Y 611.395,Z 977.53,A -85,B 0,C 180,E1 7628.169,E2 7628.169} C_VEL
LIN {X 0,Y 611.487,Z 977.53,A -85,B 0,C 180,E1 7634.175,E2 7634.175} C_VEL
LIN {X 0,Y 611.597,Z 977.53,A -85,B 0,C 180,E1 7640.006,E2 7640.006} C_VEL
LIN {X 0,Y 611.742,Z 977.53,A -85,B 0,C 180,E1 7644.307,E2 7644.307} C_VEL
LIN {X 0,Y 611.81,Z 977.53,A -85,B 0,C 180,E1 7648.574,E2 7648.574} C_VEL
LIN {X 0,Y 611.831,Z 977.53,A -85,B 0,C 180,E1 7652.833,E2 7652.833} C_VEL
LIN {X 0,Y 611.593,Z 977.53,A -85,B 0,C 180,E1 7657.656,E2 7657.656} C_VEL
LIN {X 0,Y 611.542,Z 977.53,A -85,B 0,C 180,E1 7662.878,E2 7662.878} C_VEL
LIN {X 0,Y 611.486,Z 977.53,A -85,B 0,C 180,E1 7667.292,E2 7667.292} C_VEL
LIN {X 0,Y 611.345,Z 977.53,A -85,B 0,C 180,E1 7671.819,E2 7671.819} C_VEL
